# B&R Automation Studio project TD52 (part 130)

#### op_stateCyclic.st - OpState task
```iecst
(*******************************************************************************
AGGR: selection of the operating state (cyclic)

This code is confidential AND proprietary to the INNIO Company.
It may not be used in any form, or reproduced in any manner, without the express
written permission of the INNIO Company.
Copyright, INNIO Company, 2023

Customized modifications: -
------------------------
- Calculation of actual power in kW and permill
- Filtering of actual power
- Selection of the operating state of the engine in dependence of
  speed (n_ist) generator switch (gen_sch) and mains switch (net_sch)
- Creating of operating message for the alarmmanagement

History:
-------
V0.1	13-06-2001	Fahringer, generated from betr_zus V0.2
		20-07-2001	Fahringer, last modification
V0.2	03-09-2002	Fahringer, clculation of n_ist, p_ist, P_IST_OF,
							   ssPowerEx, P_IST_PROM add
V0.3	26-10-2002	Fahringer, engine speed meassured via ignition system
V0.31	21-11-2003	Fahringer, 100 rpm hystersis between StartM and LeerlM
V0.4	18-04-2004	Fahringer, calculation of speed is done in eng_ctr
V0.5	12-02-2007	Weitzer,   copy DIs for GCB and MCB to existiong PVs
							   replace mA power input by ssPAct from MMUSynch
V0.51	18.01.2008	Lechner,   adapted net_sch for test-bench run
V0.52	30.09.2010	Maier (BuR),	allocation DI_GCB_ON_TC1 to gen_sch deleted
		30.09.2010	Maier (BuR),	gen_sch replaced with GCB_ON_TC1
		01.10.2010	Maier (BuR), 	net_sch replaced with bPowerMode
		01.10.2010	Maier (BuR),	DI_MCB_ON_TC1 replaced with MCB_ON_TC1

--------------------
V3.99.0	19.10.2011	Graus,		implementation of the module for modular software
V3.99.1	24.10.2012	Graus,		extension of early opening of gas valves
V3.99.2	07.11.2012	Graus,		upgrade opstate machine function
								start state only is activated in transition from stop state
V3.99.3	12.11.2012	Graus,		change PT of xTOF_OpHour to T#10s
					Ze			AND NOT M_ABLOCK; 	 *changed, 4.6.13*
		18.11.2013	Graus,		bugfix FOR possible division BY 0
		17.12.2013	Graus,		bugfix - use case for OMSS and RSS state instead of direct comparisons in logic terms
V3.99.4 29.01.2014 	zengerer	bGV_Start_ScaveBlock Interface
V4.00.0 11.02.2014 	Graus,		change Version TO 4.0
V4.00.1 06.03.2014 	Graus,		change name of bGlowIgnPrevent to bGlowIgnPrevActive
V4.00.2 30.04.2014	Graus, Ze	M_ABLOCK := NOT(
V4.01.0 19.05.2014  Denk		Bugfix. Abstellstörung 1023 wie bei XT4 Pilotanlage
								Blockierung mit N_OP.tDI_Dem_EU_Block.Di
V4.01.1 27.05.2014  Graus		Delay FOR OMSS states like in XT3 (T=1s)
								Bugfix FOR bEng_Bloc
V4.01.2 27.05.2014  Graus		add bLockAckStarter to blocking engine
V4.01.3 02.06.2014	Weitzer		logic of M_ABLOCK corrected
					Denk/Weitzer block engine by EVU corrected
V4.01.4 24.06.2014  Graus		add bEng_Bloc_SGM(M_GM_Ref) to opstate logic
V4.01.5	15.10.2014	Caks,		added glow ignition, blocks module after run
V4.01.6	27.11.2014	Graus,		add submode TO opstate status
V4.02.0	24.02.2015	Graus,		add changes for J920 blocking engine
V4.02.1 13.03.2015	Graus,		bugfix: invert usage of IN_OP.bEng_Bloc_EC for bEng_Bloc
		20.10.2015	Caks,		added counters for: demand, netp and island operation
V4.03BETA 15.12.	Zengerer	new State 32: waiing for next automatic start (for new BR4 start procedure)
V4.03	26.01.2016	Perktold	changed bEng_Block_EVU in case of manual mode
V4.04.00	11.10.2016	Gwiggner	change Version TO 4.04
			19.10.2016	Gomez Ortiz	Modification of the cooling run phase
			28.10.2016	Gomez Ortiz	Separation between engine operation hour counter and unit op. hour counter
			21.12.2016  Denk		Modification for WinMOD simulation

 			02.02.2016	Zengerer	Modification for state 32 waiting for next automatic start
 			02.02.2017	lettenb.	OUT_OP.bEng_Bloc: ...FC_Rdy included(sky)
V4.05.00	24.04.2017	Denk		SWAT 920 Rel.2, block engine after 5 times W2462
			10.05.2017	Gomez Ortiz	Changes for Spezifikation_Ölkreislauf_Schnellstart_BR9
			14.06.2017	lettenb.	ZM_M_REL: bRelEngStart_OilSkid added acc.spec.gen.oilskid, xGR_MAXR_OpenGV.Gw:= 80->60 for 920(fahringer)
			26.06.2017	lettenb.	tEng_Aux_Dem_CDR2/3 added for multiple use(grain)
			10.07.2017	Denk		SWAT 920 Rel.3, block engine after 5 times W2465
			31.07.2017  Denk		SWAT 920, changes after validation. Deflagration protection different function for type 6 and type 9
			07.11.2017  Perktold,	op_state Task changed for houseload requirement
			19.01.2018	Gomez Ortiz	Extension of the early open valve timing for type 9 engines
			09.02.2018	Perktold	920er FastStart change for OUT_OP.tEng_Aux_Dem_CDR.Do calculation - bFS_Act deleted
V4.05.02	05-04-2018	Perktold,	added IN_OP.bFS_Act for OilSkid Start Release Type 9
V4.05.03	05-09-2018	Gwiggner	BU 01: bugfix function block xTP_OpenGV
V4.06.00	12-06-2018	Perktold	changes for GEN2/FastStart
V4.06.01	18.09.2018	Zengerer	new engine blocking at W1995 Perm Error
			03-10-2018	Hohensinner	Bugfix: Engine ready remote only when synchronization selector switch in position automatic
V4.07.00	25.04.2018	lettenb.	1165,9214 start lockout added, SWAT920/5
			14.01.2019	Schmid		W9249 (deflagration detection) blocks engine restart
V4.07.01	30.01.2019	Hohensinner	Code clean up and Diagnose Interfaces
			03.02.2019	Perktold	tEng_Run.Do geändert (BugFix)
			25.02.2019	lettenb.	bERV_NotRdy added, engine room ventilation not ready - block engine start, PWR-FFI-2018-0637 gem. TA 1100-0110
			13.03.2019	Hohensinner	block engine at low EO/ECW temperatures for type9, block engine at grid code data structure failure
V4.07.04	10.04.2019	Hohensinner	removed UPS DI signals from engine blocked array & cleanup #07
V4.07.05	15.05.2019	Hohensinner	added EngBlock_PlantCtr DI --> Blocks module smooth
			20.05.2019	Hohensinner	EngBlock_PlantCtr DI debugged for smooth shutdown in manual mode
			04.11.2019	Schmidt		BU 01: Type 6 cooldown run duration modified from 0s to 10s
V4.09.00	28.11.2019	lettenb.	bBloc_SY_ProtTest added, protection test(ThJ)
			13.01.2020	Arnold,		time delay for early GV opening changed to 9.8s
			12.02.2020	Zuschnig, 	included B2972 and B2973 - Power Mode on/off
V4.10.00	22.05.2020	lettenb.	bEng_Bloc[29-33] added
			20.10.2020	Zuschnig,	removed activation of module blocked by oil skid only if fast start is active -> always active
			16.10.2020	Weitzer,	release power mode by customer bit bReq_PowMod_Ext
			07.10.2020	Perktold	added fast start counter
			18.01.2021	Perktold	unbundling emergency stop and fire alarm
			18.01.2021	Weitzer		IN_OP.bBloc_SY_Rel_Cust to SY release array added
			27.01.2021  Zuschnig	Ensure TON,TOF,TP are always executed
V4.11.00	22.11.2021	Perktold,	added myPlant remote request/P-setpoint
			14.10.2021	Andre,		added SAFI in operation mode to start up release
			02.02.2022	Schmid,		no start blockade by ECWP_FC_Rdy in case of black start
V4.12.00	08.09.2022	Andre,		added SEMIC in operation mode to start up release
			20.09.2022	Perktold,	Additional delay for ignition deactivation for non-successful starts
			26.09.2022	Perktold,	Added IN signal to xTOFIgn_Dem in case of a prio 1 trip
			10.01.2023	lettenb.	bReq_Bloc[4]: bOMSS_MAN->(OUT_OP.iIdx_OMSS = 1), bOMSS_MAN is too slow for bumpless switchover MAN -> AUT, #966
			25.01.2023	Tinello		Added engine blocked by charge temperature after TC
V4.13.00	26.09.2023	Farre,		Addition engine blocked by LCB opened (info #37)
			24.08.2023	Zengerer	Add counter correction IN_OP.iCnt_OpHours_Set, iCnt_UnitOpHours_Set, iCnt_FastStarts_Set, iCnt_FastStarts_Set
			03.11.2023	Zuschnig	Add operating counter low load
			20.11.2023	Farre,		added "request power mode" interface from CU needed for Microgrid (2023-168)
			04.12.2023	Goenczi		Added Emergency request via Bus coupling - bEng_Dem_EPS_Bus
			04.12.2023	Goenczi		Hand over iIdx_Eng_State to OUT_OP
			17.01.2024	Schmidt		Bugfix deflagration protection: added IN_OP.bIgnDeflPrct_Off to ignition demand logic (issue 1406)
V4.14.00	28.03.2024	Soto/Farre,	Added CAN WG configuration for start up release (2023-174)
			25.10.2024	Farre		include in bEng_Bloc[1] - rel. sync- when GCB position signal failure and enigne stopped (2024-241)
			25.11.2024	Bacci		T6 Start procedure with purge start (2024-219): added waiting time for starter release in state 32 and 7

Instructions for use:
--------------------

Outstandings:
------------

*******************************************************************************)

FUNCTION AND_Array
	memcpy(ADR(Arrayx),Adress,MIN(40,Size) + 1);
	AND_Array	:=	 TRUE;
	FOR i:= 0 TO MIN(40,Size) DO
		AND_Array	:=	AND_Array AND Arrayx[i];
	END_FOR
END_FUNCTION

FUNCTION OR_Array
	memcpy(ADR(Arrayx),Adress,MIN(40,Size) + 1);
	OR_Array	:=	 FALSE;
	FOR i:= 0 TO MIN(40,Size) DO
		OR_Array	:=	OR_Array OR Arrayx[i];
	END_FOR
END_FUNCTION

FUNCTION DINT_INC_CNT
	DINT_INC_CNT	:=	Input + 1;
	IF DINT_INC_CNT >= 1000000000 THEN
		DINT_INC_CNT := DINT_INC_CNT - 1000000000;		(* check upper limit *)
	ELSIF DINT_INC_CNT <= -1000000000 THEN
		DINT_INC_CNT := DINT_INC_CNT + 1000000000;		(* check lower limit *)
	END_IF;
END_FUNCTION

PROGRAM _CYCLIC

(** 1: Execute EngType for Module *)
	xEngType.Motortype := INT_TO_UINT(Para.iEng_Motortype);
	xEngType();

(** 2: Build OMSS and RSS bits for states *)
	xTOF_OFF(IN := OUT_OP.iIdx_OMSS = 0, PT := T#1s);
	xTOF_MAN(IN := OUT_OP.iIdx_OMSS = 1, PT := T#1s);
	xTOF_AUTO(IN := OUT_OP.iIdx_OMSS = 2, PT := T#1s);
	xTOF_TEST(IN := OUT_OP.iIdx_OMSS = 3, PT := T#1s);
	xTOF_SCAV(IN := OUT_OP.iIdx_OMSS = 4, PT := T#1s);
	xTON_Eng_SU_Aut(IN := OUT_OP.bEng_SU_Aut, PT := T#6s);  (*V4.04 -> State 32*)

	bOMSS_OFF := xTOF_OFF.Q;
	bOMSS_MAN := xTOF_MAN.Q;
	bOMSS_AUTO := xTOF_AUTO.Q;
	bOMSS_TEST := xTOF_TEST.Q;
	bOMSS_SCAV := xTOF_SCAV.Q;

	bRSS_OFF := OUT_OP.iIdx_RSS = 0;
	bRSS_ON  := OUT_OP.iIdx_RSS = 1;
	bRSS_REM := OUT_OP.iIdx_RSS = 2;

	OUT_OP.tOMSS_MAT.Do := bOMSS_MAN OR bOMSS_AUTO OR bOMSS_TEST;

(** 3: Reject to house load type 6 / Fangen im Eigenbedarf Baureihe 6*)
	bTrigger_Island	:= xEngType.Type6 AND Para.bRej2houseload AND xOpMode.NetP AND (IN_OP.rN_EngAct >= rN_Eng_Limit);
	TOF_bTrigger_Island(IN := bTrigger_Island, PT := tOff_Trigger);

(** 4: Powermode *)
	bPowerMode := ((IN_OP.tMCB_On.Di AND NOT TOF_bTrigger_Island.Q) AND (IN_OP.tMnsOk.Di OR NOT IN_OP.bTestBenchModeIsland)) OR IN_OP.bReq_PowMod OR IN_OP.bReq_PowMod_Ext;

	IF IN_OP.tGCB_On.Di AND OUT_OP.tEng_Run.Do AND NOT IN_OP.tMCB_On.Di AND NOT IN_OP.bMCB_DemSy AND (IN_OP.bReq_PowMod OR IN_OP.bReq_PowMod_Ext) AND NOT bMsg2973 THEN
		bMsg2972 := TRUE;
	ELSE
		bMsg2972 := FALSE;
	END_IF;

	TOF_b2973(IN := EDGENEG (bMsg2972), PT := T#5s);
	bMsg2973 := TOF_b2973.Q;

(** 5: OpMode State machine: condition of engine state in dependence of actual speed, generator switch and mains switch*)
	IF IN_OP.rN_EngAct < 50 THEN							(* condition for engine operating state STOP	*)
		OUT_OP.iSt_OpMode := 16#00010000 * 10;	(* StopM -> 10 *)
	ELSE
		IF xOpMode.Stop THEN (* transition from stop mode *)
			bStop2Start := TRUE;
		END_IF;
		IF (IN_OP.rN_EngAct < Para.rN_Start_Trig) AND bStop2Start THEN			(* condition for engine operating state START	*)
			OUT_OP.iSt_OpMode := 16#00010000 * 30;	(* StartM -> 30 *)
		ELSE
			bStop2Start := FALSE;
			IF IN_OP.tGCB_On.Di AND bPowerMode THEN		(* condition for engine operating in parallel with system	*)
				OUT_OP.iSt_OpMode := 16#00010000 * 50;	(* NetpM -> 50 *)
			ELSE
				IF IN_OP.tGCB_On.Di AND NOT bPowerMode THEN	(* condition for engine operating in isolated mode	*)
					OUT_OP.iSt_OpMode := 16#00010000 * 60;	(* InselM -> 60 *)
				ELSIF IN_OP.rN_EngAct >= Para.rN_Start_Trig THEN
					OUT_OP.iSt_OpMode := 16#00010000 * 40;	(* LeerlM -> 40 *)
				END_IF;
			END_IF;
		END_IF;
	END_IF;

	xOpMode(in := OUT_OP.iSt_OpMode);

(** 6: Emergency Request *)
	OUT_OP.bEng_Dem_EPS	:=
							((IN_OP.tEng_Dem_EPS_Ext.Di OR IN_OP.bEng_Dem_EPS_Bus OR IN_OP.bEng_Dem_EPS_Sy) AND NOT IN_OP.bOnly_Island)
						OR 	(IN_OP.bOnly_Island AND NOT IN_OP.bOtherGenParallel);

	xTOF_EngDemEPS(IN:= OUT_OP.bEng_Dem_EPS AND NOT IN_OP.tGCB_On.Di, PT:= T#60s);
	bNoMon4BlackStart := xTOF_EngDemEPS.Q AND OUT_OP.bEng_Dem_EPS; //T14

(** 7: Excitation bit *)
	OUT_OP.bEng_SUpE := IN_OP.tEng_SUExc_Rel.Di;

(** 8: Plant control *)
	(** 8.1: W1188 release by station missing *)
	xTP_AT27(IN := NOT IN_OP.tRel_MasCtr.Di, PT := T#300s);
	AT27	:=	NOT xTP_AT27.Q AND IN_OP.tRel_MasCtr.Di;

	(** 8.2: Wxxxx block by plant control - smooth *)
	xTON_Block_PlantCtr(IN:= IN_OP.tEngBlock_PlantCtr.Di AND IN_OP.tEngBlock_PlantCtr.GoodQual, PT:=T#100ms);
	bEng_Block_PlantCtr	:=	xTON_Block_PlantCtr.Q;

	IF bEng_Block_PlantCtr AND bOMSS_MAN THEN																	(* set load to zero in manual mode *)
		VIS2MM.rP_set_vis		:=	0;
	END_IF
	IF EDGEPOS(bEng_Block_PlantCtr AND bOMSS_MAN AND (OUT_OP.rP_Act_Norm_Filt < 0.1 OR xOpMode.Island)) THEN	(* stop engine if under 10% load or island mode *)
		OUT_OP.bEng_Stop_Man	:=	TRUE;
	END_IF

(** 9: Engine Blocked Array  *)
	(* Info compared to old SW: 0-7 represents old variable "NOT ZM_M_REL" *)
	bEng_Bloc[0]	:=	NOT ((IN_OP.bMainsReturn AND (IN_OP.bRelMainsConnect OR xOpMode.NetP)) OR IN_OP.bRel_Island OR IN_OP.bRel_IslandAfMITime OR NOT Para.bSyActive);	(* Mains failure *)
	bEng_Bloc[1]	:=	(NOT IN_OP.bRelEngOpFromSy) OR IN_OP.bGCB_psf_EngStop;																								(* Release from Sync missing or gcb position failure when engine stopped *)
	bEng_Bloc[2]	:=	NOT AT27 OR (bEng_Block_PlantCtr AND NOT bEng_StaSpdExc);																							(* W1188 release by station missing *)
	bEng_Bloc[3]	:=	NOT IN_OP.bGasSupplyOk;																																(* Gas supply missing *)
	bEng_Bloc[4]	:=	NOT (	(NOT xEngType.Type9 AND NOT IN_OP.bDeflagrationPrct)																						(* Deflagration protection not Type 9 *)
							OR	(xEngType.Type9 AND ((NOT IN_OP.bDeflagrationPrct AND NOT IN_OP.bPBC_Active) OR IN_OP.bPBC_Active)));										(* Deflagration protection Type 9 *)
	bEng_Bloc[5]	:=	NOT IN_OP.tGV_Rel.Do;																																(* Gas valve release missing *)
	bEng_Bloc[6]	:=	IN_OP.bLockAckStarter;																																(* Starter temperature *)
	bEng_Bloc[7]	:=	xEngType.Type9 AND NOT bEng_StaSpdExc AND NOT IN_OP.bRelEngStart_OilSkid;																			(* Oil skid Type 9 *)
	bEng_Bloc[8]	:=	IN_OP.bEng_Block_Customized;																														(* Customer specific *)
	bEng_Bloc[9]	:=	IN_OP.tMCB_On.Di AND NOT OUT_OP.tEng_Run.Do AND IN_OP.tP_GenC_Bloc.Do;																				(* EU - Power reduction over limit *)
	bEng_Bloc[10]	:=	(IN_OP.bMsg3583 OR 	IN_OP.bMsg3584) AND Para.bGlowIgnPrevActive;																					(* Special gas: Exhaust gas temperatures *)
	bEng_Bloc[11]	:=	IN_OP.bSG_Eng_Block_EGT; 																															(* Special gas: blocked after 30min operation *)
	bEng_Bloc[12]	:=	IN_OP.bEng_Bloc_EC;(* AND Para.bSA_PI_Active;*)																										(* Blocked by Engine Controller*)
	bEng_Bloc[13]	:=	IN_OP.bSAFIPBCConfNotOK AND Para.bSA_PBC_Active;																									(* Blocked by SAFI PBC configuration *)
	bEng_Bloc[14]	:=	(bOMSS_AUTO AND NOT bEng_StaSpdExc AND NOT IN_OP.tScavFanFC_Rdy.Di);																				(* Blocked by FC scavanging fan *)
	bEng_Bloc[15]	:=	(bOMSS_AUTO AND NOT bEng_StaSpdExc AND NOT IN_OP.tECWP_FC_Rdy.Di AND NOT bNoMon4BlackStart);														(* Blocked by FC ECWP *)
	bEng_Bloc[16]	:=	(bOMSS_AUTO AND NOT bEng_StaSpdExc AND NOT IN_OP.tEOP_FC_Rdy.Di);																					(* Blocked by FC EOP *)
	bEng_Bloc[17]	:=	(bOMSS_AUTO AND NOT bEng_StaSpdExc AND NOT IN_OP.tBbBlower_FC_Rdy.Di);																				(* Blocked by FC Byblower *)
	bEng_Bloc[18]	:=	((IN_OP.bAMM_Pr_MGT_a_Filt_BlockStart OR IN_OP.bAMM_Pr_PCGT_a_Filt_BlockStart) AND xEngType.Type9); 												(* 5times MSF in gastrain *)
	bEng_Bloc[19]	:=	(IN_OP.bMsg9214 AND NOT bEng_StaSpdExc AND xEngType.Type9); //SWAT920/5																				(* Engine turn equipment active *)
	bEng_Bloc[20]	:=	(IN_OP.bMsg1165 AND NOT bEng_StaSpdExc AND xEngType.Type9); //SWAT920/5																				(* Exhaust gas scavanging failure *)
	bEng_Bloc[21]	:=	(IN_OP.bMsg1995 AND NOT bEng_StaSpdExc );																											(* Perm failure in stop mode *)
	bEng_Bloc[22]	:=	IN_OP.tMCB_On.Di AND NOT OUT_OP.tEng_Run.Do AND IN_OP.tDI_Dem_EU_Block.Di;																			(* EU - Blocked by DI *)
	bEng_Bloc[23]	:=	IN_OP.tMCB_On.Di AND NOT OUT_OP.tEng_Run.Do AND IN_OP.bEng_Block_EVU;																				(* EU - Blocked by Bus *)
	bEng_Bloc[24]	:=	IN_OP.bMsg9249 AND NOT bEng_StaSpdExc;																												(* Deflagration detection *)
	bEng_Bloc[25]	:=	IN_OP.bERV_NotRdy AND NOT bEng_StaSpdExc;																											(* engine room ventilation not ready *)
	bEng_Bloc[26]	:=	xEngType.Type9 AND bOMSS_MAN AND NOT bEng_StaSpdExc AND IN_OP.bMsg2524;																				(* Type9: EO Temp low *)
	bEng_Bloc[27]	:=	xEngType.Type9 AND bOMSS_MAN AND NOT bEng_StaSpdExc AND bT_ECW_Lo;																					(* Type9: ECW Temp low *)
	bEng_Bloc[28]	:=	IN_OP.bEng_Bloc_GR AND NOT bEng_StaSpdExc;																											(* GR - data structure failure *)
	bEng_Bloc[29]	:=	NOT IN_OP.tScavFanCB_trip.Di AND NOT bEng_StaSpdExc;																								(* Blocked by CB scavenging fan tripped *)
	bEng_Bloc[30]	:=	NOT IN_OP.tGenIF_CB_On.Di AND NOT bEng_StaSpdExc;																									(* Blocked by CB generator interface panel tripped *)
	bEng_Bloc[31]	:=	IN_OP.bAMM_OilSkid_PumpLP_CB AND NOT bEng_StaSpdExc AND xEngType.Type9;																				(* Type9: Blocked by CB oil skid LP oil pump tripped *)
	bEng_Bloc[32]	:=	IN_OP.bAMM_OilSkid_PumpHP_CB AND NOT bEng_StaSpdExc AND xEngType.Type9;																				(* Type9: Blocked by CB oil skid HP oil pump tripped *)
	bEng_Bloc[33]	:=	IN_OP.bAMM_OilSkid_MCB AND NOT bEng_StaSpdExc AND xEngType.Type9;																					(* Type9: Blocked by oil skid main switch auxiliaries opened *)
	bEng_Bloc[34]	:=	NOT IN_OP.tECWP_CB_On.Di AND NOT bEng_StaSpdExc;																									(* Blocked by CB ECWP tripped *)
	bEng_Bloc[35]	:=	IN_OP.bEngBloc_EX AND NOT bEng_StaSpdExc;
	bEng_Bloc[36]	:=	NOT IN_OP.bRelEngStart_Ch_T2 AND NOT bEng_StaSpdExc;																								(* Blocked by charge temperature after TC *)
	bEng_Bloc[37]	:=	NOT IN_OP.tLineCB_On.Di AND IN_OP.tLineCB_On.GoodQual;																								(* Blocked by line circuit breaker open *)
	bEng_Bloc[38]	:=	IN_OP.bBlock_WG_CAN_Conf;																															(* Blocked by wastegate configuration in progress *)

	OUT_OP.bEng_Bloc		:=	OR_Array(ADR(bEng_Bloc),50);	(* 1 = engine is blocked *)
	MM2VIS.bEng_Bloc		:=	bEng_Bloc;						(* Array to VIS *)
	MM2VIS.bEng_Bloc_Show	:=	(iIdx_Eng_State = 19);			(* Show Array only on HMI if engine is blocked *)

(** 10: Demand Auxiliaries  *)
	OUT_OP.bEng_Aux_Dem :=	(OUT_OP.bEng_Dem AND (IN_OP.bPurgeER_Rdy OR NOT Para.bPurgecycle_Active) AND (IN_OP.bEGScav_Rdy OR OUT_OP.bEng_Dem_EPS)) OR IN_OP.bGV_On;

(** 11: Release Engine *)
	OUT_OP.bEng_Rel :=	OUT_OP.tOMSS_MAT.Do
						AND ((NOT (bGnlTrip1 OR bGnlTrip2 OR bGnlTrip3)) OR bDryTestBench)
						AND IN_OP.tPB2MM.bParaSetupOk;

(** 12: Start Up Release - Array for Manual and Automatic Mode *)
	bEng_SU[0]	:=	OUT_OP.bEng_Rel;																		(* Engine released *)
	bEng_SU[1]	:=	NOT bEng_StaSpdExc;																		(* Start speed not exceeded *)
	bEng_SU[2]	:=	IN_OP.bRelEngOp_Aux;																	(* Release from Auxiliaries *)
	bEng_SU[3]	:=	IN_OP.bScavFinished;																	(* Scavanging finished *)
	bEng_SU[4]	:=	(IN_OP.bPurgeER_Rdy AND IN_OP.tRel_ER_PurgeCycle.Di) OR NOT Para.bPurgecycle_Active;	(* Purge finished *)
	bEng_SU[5]	:=	NOT IN_OP.bEng_Bloc_SGM;																(* Special gas mixer calibration routine not active *)
	bEng_SU[6]	:=	IN_OP.bIC_OperationState AND IN_OP.bSA_CfgDone;											(* SEMIC used and in operation state *)

	MM2VIS.bEng_SU			:=	bEng_SU;																	(* Array to VIS *)
	MM2VIS.bEng_SU_Show		:=	(iIdx_Eng_State = 32) OR (iIdx_Eng_State = 9) OR (iIdx_Eng_State = 8) OR (iIdx_Eng_State = 6);	(* Show Array only on HMI if in this states *)

(** 13: Engine Ready Manual Mode *)
	OUT_OP.bEng_Rdy_Man :=	OUT_OP.bEng_Rel AND bOMSS_MAN AND NOT bEng_StaSpdExc AND NOT OUT_OP.bEng_Bloc;

(** 14: Start Impulse 10s long *)
	xTP_Imp_Start(IN := IN_OP.bEng_Start, PT := T#10s);
	OUT_OP.bImp_Start := xTP_Imp_Start.Q;

(** 15: Delay next manual start for 5s *)
	xTOF_BlocDelay_ManStart(IN := OUT_OP.bImp_Start OR IN_OP.bEng_Start , PT := T#5s);
	OUT_OP.bBlocDelay_ManStart := xTOF_BlocDelay_ManStart.Q;

(** 16: Blocking demand for 30s after a Start *)
	xTOF_ANFBLO(IN := bEng_StaSpdExc, PT := T#30s);
	OUT_OP.bEng_Dem_Bloc := xTOF_ANFBLO.Q;

(** 17: Start Up Failure - Manual Mode *)
	OUT_OP.bEng_Dem_Man_SUpF :=
							(bStart OR ZM_H_ANF OR OUT_OP.bEng_Dem_Aut OR (bOMSS_AUTO AND OUT_OP.bEng_CDR))
						AND OUT_OP.bEng_Rel
						AND bOMSS_MAN
						AND NOT OUT_OP.bEng_Stop_Man
						AND NOT OUT_OP.bEng_Bloc;

	ZM_H_ANF :=				OUT_OP.bEng_Dem_Man_SUpF
						AND (NOT OUT_OP.bEng_Dem_Bloc OR IN_OP.bGV_On OR IN_OP.bEng_Start);

(** 18: Engine Demand - Manual Mode *)
	OUT_OP.bEng_Dem_Man :=
						(NOT bStart OR OUT_OP.bEng_Dem_Man)
						AND ZM_H_ANF;

(** 19: Start Up Release - Manual Mode *)
	OUT_OP.bEng_SU_Man	:=	AND_Array(ADR(bEng_SU),6) AND OUT_OP.bEng_Dem_Man;			(* 1 = start up *)

(** 19: Engine Start up - Manual Mode *)
	OUT_OP.bEng_Rel_SU	:=	OUT_OP.bEng_SU_Man AND (NOT OUT_OP.bBlocDelay_ManStart OR IN_OP.bEng_Start);

(** 20: Notstrom Anforderung ohne reine Inselanlagen *)
	bRequest_EPS	:=	OUT_OP.bEng_Dem_EPS AND NOT IN_OP.bOnly_Island;				(* EPS *)

(** 21: Engine automatic request *)
	(** 21.1: Engine in Automatic demanded *)
	bReq_Dem[0]		:=	bRSS_ON;																	(* ON *)
	bReq_Dem[1]		:=	bRSS_REM AND VIS2MM.bRemoteReq AND Para.bRemoteReqActive;					(* HMI Button *)
	bReq_Dem[2]		:=	bRSS_REM AND IN_OP.tReq_PeakLoad.Di;										(* DI - Peakload *)
	bReq_Dem[3]		:=	bRSS_REM AND IN_OP.bBus_Dem;												(* BUS *)
	bReq_Dem[4]		:=	bRSS_REM AND IN_OP.bEngDSS_Mains;											(* Mains control *)
	bReq_Dem[5]		:=	bRSS_REM AND IN_OP.bCust_Dem;												(* Demand from Custom Module *)
	bReq_Dem[6]		:=	bRSS_REM AND IN_OP.tDemEngOpExt.Di;											(* DI - ExtDem *)
	bReq_Dem[7]		:=	bRSS_REM AND VIS2MM.bRemoteReq_myPlant AND Para.bRemoteReqMyPlantActive;	(* myPlant *)

	bReq_Remote		:= bReq_Dem[1] OR bReq_Dem[7];													(* Engine Demand via remote (HMI or myPlant) *)

	bRequest_Dem	:=	OR_Array(ADR(bReq_Dem),7);
	MM2VIS.bReq_Dem		:=	bReq_Dem;
	MM2VIS.bReq_Dem_Show:=	TRUE;		(* not used at moment *)

	(** 21.2: Block Automatic Engine demand *)
	bReq_Bloc[0]	:=	IN_OP.bGT_DemRelGasTypSwh; 									(* Gas type switching *)
	bReq_Bloc[1]	:=	IN_OP.tP_GenC_Bloc.Do;										(* EU load reduction > limit *)		//EVU_BLOCK_INT	Mathias 2.6.2014
	bReq_Bloc[2]	:=	IN_OP.tDI_Dem_EU_Block.Di;									(* EU - DI *)						//DI_EVU_BLOCK  Mathias 2.6.2014
	bReq_Bloc[3]	:=	IN_OP.bEng_Block_EVU;										(* EU - Bus *)
	bReq_Bloc[4]	:=	bRequest_EPS AND (OUT_OP.iIdx_OMSS = 1);					(* EPS & OMSS Man *)
	bReq_Bloc[5]	:=	bRequest_EPS AND IN_OP.bSmoothDischarge;					(* EPS & smooth discharge *)
	bReq_Bloc[6]	:=	bEng_Block_PlantCtr;										(* PlantCtr *)

	bRequest_Bloc	:=	OR_Array(ADR(bReq_Bloc),6);
	MM2VIS.bReq_Bloc:=	bReq_Bloc;
	MM2VIS.bReq_Bloc_Show	:=	TRUE;	(* not used at moment *)

	(** 21.3: Request Engine - M_ANF *)
	xTON_T105(IN := bOMSS_TEST AND (xTON_T105.Q OR OUT_OP.tEng_Run.Do), PT := T#300s);	(* Test delay *)

	bReq_A[0] 		:=	bRequest_Dem AND NOT bRequest_Bloc;								(* Requested and not blocked *)
	bReq_A[1] 		:=	bRequest_EPS AND NOT IN_OP.bSmoothDischarge AND NOT bOMSS_MAN AND NOT bEng_Block_PlantCtr;	(* EPS request *)
	bReq_A[2] 		:=	bOMSS_MAN AND IN_OP.tGCB_On.Di;									(* OMSS Man and GCB closed *)
	bReq_A[3] 		:=	bOMSS_TEST AND (NOT xTON_T105.Q OR IN_OP.tReq_Test.Di); 		(* OMSS Test and Test Delay / DI *)

	bRequest_A 		:=	OR_Array(ADR(bReq_A),3);
	MM2VIS.bReq_A	:=	bReq_A;
	MM2VIS.bReq_A_Show	:=	bOMSS_AUTO;

	M_ANF	:= 	bRequest_A; 	(* rückwärtskompatiblität *)

(** 22: Engine demand start up failure & Engine demand in automatic mode *)
	xGRMinR_KWT(Gw := Para.rT_ECW_LimLo, Hy := Para.rT_ECW_HyLo, In := IN_OP.tT_ECW.Ai);
	xTON_kwtp(IN := xGRMinR_KWT.Q AND IN_OP.tPB2MM.bParaSetupOk, PT := T#2s);
	bT_ECW_Lo := xTON_kwtp.Q;	(* entspricht AN_KTMI - Kühlwassertemperatur minimum *)									//Überprüfen ob in powersel unten benötigt, vllt besser: von HC hermappen

	(* Release automatic start - M_ABLOCK *)
	bEng_Dem_A[0]	:=	NOT bT_ECW_Lo OR OUT_OP.bEng_Dem_EPS; 														(* Engine cooling water temperature not low *)
	bEng_Dem_A[1]	:=	NOT IN_OP.bPr_N2_LoTon OR OUT_OP.tEng_Run.Do OR IN_OP.bGT2_Select OR NOT IN_OP.bRel_ScavN2;	(* N2 scavanging done *)
	bEng_Dem_A[2]	:=	NOT OUT_OP.bEng_Bloc;																		(* Engine not blocked *)

	(* Release automatic start - OUT_OP.bEng_Dem_Aut_SUpF *)
	bEng_Dem_A[3]	:=	OUT_OP.bEng_Rel;																			(* Engine released *)
	bEng_Dem_A[4]	:=	bOMSS_AUTO OR bOMSS_TEST;																	(* OMSS Auto or Test *)
	bEng_Dem_A[5]	:=	bRequest_A;																					(* Engine automatic start requested *)

	(* Release automatic start - OUT_OP.bEng_Dem_Aut*)
	bEng_Dem_A[6]	:=	NOT bEng_StaSpdExc OR IN_OP.bGV_On OR IN_OP.bEng_Start;										(* Engine starts / runs *)
	bEng_Dem_A[7]	:=	NOT OUT_OP.bEng_Dem_Bloc OR	OUT_OP.tEng_Run.Do OR OUT_OP.bEng_Dem_Aut;						(* Engine request blocked, before: M_ANFBLO *)
	bEng_Dem_A[8]	:=	NOT IN_OP.tERDF_BLOCK.Do;																	(* ERDF *)
	bEng_Dem_A[9]	:=	NOT IN_OP.bOpMsg_Plim_ERDF_ABF_SOnOf;														(* Load reduction over limit *)

	M_ABLOCK					:=	AND_Array(ADR(bEng_Dem_A),2); 	//M_ABLOCK wird nun im array gebildet, bildet sich nur aus 0 bis 2
	OUT_OP.bEng_Dem_Aut_SUpF	:=	AND_Array(ADR(bEng_Dem_A),5);	//OUT_OP.bEng_Dem_Aut_SUpF bildet sich nur aus 0 bis 5
	OUT_OP.bEng_Dem_Aut			:=	AND_Array(ADR(bEng_Dem_A),9);
	MM2VIS.bEng_Dem_A			:=	bEng_Dem_A;
	MM2VIS.bEng_Dem_A_Show		:=	bOMSS_AUTO;

	ZM_M_BERAUT :=			OUT_OP.bEng_Rel
						AND (bOMSS_AUTO OR (bOMSS_TEST AND OUT_OP.bEng_Dem_EPS));

(** 23: Engine ready for automatic mode *)
	OUT_OP.bEng_Rdy_Aut		:=	ZM_M_BERAUT AND M_ABLOCK; 	(*changed, 4.6.13*)

(** 24: Engine ready for automatic mode - info for exitation system *)
	OUT_OP.bEng_Rdy_Aut_Exc	:=	ZM_M_BERAUT	AND (bRequest_A OR NOT IN_OP.bOnly_Island);

(** 25: Engine ready for remote operation *)
	OUT_OP.tEng_Rdy_Rem.Do	:=	OUT_OP.bEng_Rdy_Aut AND bRSS_REM AND IN_OP.iIdx_SyOMSS = 2;

(** 26: Engine automatic startup *)
	OUT_OP.bEng_SU_Aut		:=	AND_Array(ADR(bEng_SU),6) AND OUT_OP.bEng_Dem_Aut;		(* 1 = start up *)

(** 27: Engine monitoring of after start for 10s *)
	xTOF_T9(IN := IN_OP.bEng_Start, PT := T#10s);
	OUT_OP.bEng_MonOff := xTOF_T9.Q;

(** 27: Engine stop in manuel mode *)
	OUT_OP.bEng_Stop_Man	:=	(OUT_OP.bEng_Rel AND bOMSS_MAN  AND bStop)
							OR	(OUT_OP.bEng_Rel AND bOMSS_MAN  AND OUT_OP.bEng_Bloc)
							OR	(OUT_OP.bEng_Rel AND bOMSS_MAN  AND NOT bEng_StaSpdExc AND IN_OP.bMaxPreLubeTime)
							OR	(OUT_OP.bEng_Rel AND bOMSS_AUTO AND IN_OP.bN_EngStartDrop)
							OR	(OUT_OP.bEng_Rel AND bIgn_DemTemp AND OUT_OP.bEng_Stop_Man);						//latch until ignition demand off

(** 28: Demand Ignition *)
	xTON_T_Z_AUS(IN := IN_OP.bMsg1026, PT := T#10s);

	bIgn_Dem[0]	:=	NOT IN_OP.bMsg1022 OR IN_OP.bIgn2_Sel;							(* A1022 - overspeed (relay)				*)
	bIgn_Dem[1]	:=	NOT bGnlTrip1 OR IN_OP.bIgn2_Sel;								(* Trip1									*)
	bIgn_Dem[2]	:=	NOT xTON_T_Z_AUS.Q;												(* A1026 - Shutdown failure, 10s delayed	*)
	bIgn_Dem[3]	:=	IN_OP.bRel_IgnOn OR bEng_StaSpdExc;								(* Release ignition from starter (AG)		*)
	bIgn_Dem[4]	:=	NOT IN_OP.bN2_ScavCoStarterOn OR NOT IN_OP.bRel_ScavN2;			(* N2 scavanging in progress				*)
	bIgn_Dem[5]	:=	NOT IN_OP.bIgnDeflPrct_Off;										(* Deflagration protection					*)

	bIgn_DemTemp	:=	AND_Array(ADR(bIgn_Dem),5) OR ((IN_OP.b_ST_DemIgn OR IN_OP.rN_EngAct <> 0) AND IN_OP.bSelfTestRunning);
	MM2VIS.bIgn_Dem	:=	bIgn_Dem;
	MM2VIS.bIgn_Dem_Show	:=	TRUE;

	(** 28.1: Demand Ignition off is delayed, only in case of priority 1 trip it is not delayed *)
	IF IN_OP.tAB2OP.bGnlTrip1 THEN
		OUT_OP.tIgn_Dem.Do := bIgn_DemTemp;
		xTOFIgn_Dem(IN:= bIgn_DemTemp);
	ELSIF NOT IN_OP.tAB2OP.bGnlTrip1 THEN
		IF bEng_StaSpdExc THEN
			xTOFIgn_Dem(IN:= bIgn_DemTemp, PT:= Ign_Dem_DelayTime);
		ELSE
			xTOFIgn_Dem(IN:= bIgn_DemTemp, PT:= Ign_Dem_DelayTime + Ign_Dem_DelayTime2);
		END_IF;
		OUT_OP.tIgn_Dem.Do := xTOFIgn_Dem.Q;
	END_IF;
	OUT_OP.bIgn_Dem	:=	OUT_OP.tIgn_Dem.Do;

(** 29: Demand gas valves *)
	(** 29.1: early opening of gas valves *)
	IF xEngType.Type9 THEN
		xGR_MAXR_OpenGV.Gw	:=	60;
		xTP_OpenGV.PT		:=	T#9s800ms;		(* Type 9 engine needs approx. 10 seconds for the ignition unit to be ready *)
	ELSE
		xGR_MAXR_OpenGV.Gw	:=	80;
		xTP_OpenGV.PT		:=	T#4s800ms;	(* Other engines need approx. 6 seconds for the ignition unit to be ready *)
    END_IF;
	xGR_MAXR_OpenGV(In := IN_OP.rN_EngAct, Hy := 10);
	xTP_OpenGV(IN:= xGR_MAXR_OpenGV.Q AND IN_OP.bEng_Start AND NOT Para.bGlowIgnPrevActive AND NOT Para.bDeAct_EarlyGV_opening AND (IN_OP.iStartCount = 1));

	(* 29.2: Release of gas valves *)
	OUT_OP.bGV_Rel :=		NOT IN_OP.bMsg1031
							AND NOT IN_OP.bMsg1054
							AND NOT IN_OP.bMsg1022
							AND NOT IN_OP.bMsg1026
							AND NOT bGnlTrip1;

	(* 29.3: Gas valves open *)
	bGV_Open[0] :=	OUT_OP.bEng_Rel OR (bGnlTrip3 AND (bOMSS_AUTO OR bOMSS_TEST));
	bGV_Open[1] :=	bIgn_DemTemp;
	bGV_Open[2] :=	IN_OP.bIgn_Run OR xTP_OpenGV.Q;
	bGV_Open[3] :=	NOT xOpMode.Stop;
	bGV_Open[4] :=	NOT OUT_OP.bEng_Stop_Man;
	bGV_Open[5] :=	OUT_OP.bGV_Rel;
	bGV_Open[6] :=	((	IN_OP.tN2_GV1_Closed.Di AND (IN_OP.tN2_GV2_Closed.Di OR NOT Para.bSel_TwoN2Valves) AND IN_OP.tScavVaClosed.Di) OR NOT IN_OP.bRel_ScavN2 OR IN_OP.bGV_On);
	bGV_Open[7] :=	NOT IN_OP.bGV_Start_ScaveBlock;	 (*new:	block gas valves from startup procedure	for scavening start *)

	OUT_OP.bGV_Open_Opstate	:=	AND_Array(ADR(bGV_Open),7);
	MM2VIS.bGV_Open			:=	bGV_Open;
	MM2VIS.bGV_Open_Show	:=	bIgn_DemTemp;

(** 30: Engine demand *)
	OUT_OP.bEng_Dem		:=	OUT_OP.bEng_Dem_Man
						OR	OUT_OP.bEng_Dem_Aut
						OR	OUT_OP.bEng_SUpE;

(** 31: RPS Demand *)
	OUT_OP.bEng_RPSDem	:=	OUT_OP.bEng_Dem
						AND NOT IN_OP.bGT_DemRelGasTypSwh
						AND (NOT bOMSS_TEST OR (bOMSS_TEST AND IN_OP.tReq_Test.Di) OR OUT_OP.bEng_Dem_EPS);

(** 32: Engine Cool down run *)
	ZM_IN_bEng_CDR	:=	OUT_OP.tEng_Run.Do
					AND ( 	((bOMSS_AUTO OR bOMSS_TEST) AND IN_OP.tGCB_On.Di)
						OR	OUT_OP.bEng_Dem_Aut
						);

	ZM_RS_bEng_CDR	:=	(NOT bOMSS_AUTO AND NOT bOMSS_TEST)
					OR	bGnlTrip1
					OR	bGnlTrip2
					OR 	OUT_OP.bEng_Bloc;

	IF xEngType.Type6 THEN
		xTOF_R_bEng_CDR(IN := ZM_IN_bEng_CDR, PT := 1000, RS := ZM_RS_bEng_CDR);  (* PT = 1000 -> Delaytime in 10ms steps -> 10s *)
	ELSIF xEngType.Type9 THEN
		xTOF_R_bEng_CDR(IN := ZM_IN_bEng_CDR, PT := 0, RS := ZM_RS_bEng_CDR);  (* PT = 0 -> Delaytime in 10ms steps -> 0s *)
	ELSE
		xTOF_R_bEng_CDR(IN := ZM_IN_bEng_CDR, PT := 6000, RS := ZM_RS_bEng_CDR);  (* PT = 6000 -> Delaytime in 10ms steps -> 6000s *)
	END_IF;

	OUT_OP.bEng_CDR := xTOF_R_bEng_CDR.Q;

(** 33: Engine run *)
	xGR_MAXR_bs_15s_rpm_hi(In := IN_OP.rN_EngAct, Gw := Para.rN_BS_Acc_LimHi, Hy := 10);
	bs_15s_rpm_hi :=
					xGR_MAXR_bs_15s_rpm_hi.Q
				AND IN_OP.tPB2MM.bParaSetupOk;
	bs_15s_rel_oper :=
					Para.bBS_Acc_Active
				AND OUT_OP.bEng_Dem_EPS
				AND OUT_OP.bEng_MonOff
				AND (bs_15s_rpm_hi OR bs_15s_rel_oper);

	IF (xOpMode.Idle OR xOpMode.Island OR xOpMode.NetP) AND NOT bN_Eng_Run THEN
		bN_Eng_Run	:= TRUE;
	ELSIF xOpMode.Stop AND bN_Eng_Run THEN
		bN_Eng_Run	:= FALSE;
	END_IF;

	OUT_OP.tEng_Run.Do :=
					OUT_OP.tOMSS_MAT.Do
				AND IN_OP.bGV_On
				AND ((bs_15s_rel_oper OR NOT OUT_OP.bEng_MonOff) OR bN_Eng_Run)	//Änderung >= rN_Start_Trig für Faststart schnellere SY
				AND (OUT_OP.bEng_CDR OR OUT_OP.bEng_Dem_Aut OR (bOMSS_MAN  AND OUT_OP.bEng_Dem_Man));

(** 34: Restart blocking *)
	xTON_RUN(IN := TRUE, PT := T#30s); (* instead RUN bit *)
	ZM_bEng_RSBoc	:=	(NOT OUT_OP.tEng_Run.Do AND xTON_RUN.Q)
					OR	EDGENEG(OUT_OP.tEng_Run.Do);

	xTP_bEng_RSBoc(IN := ZM_bEng_RSBoc, PT := T#2m);	// sinnvoller vieleicht nur auf EDGENEG gehen und das andere vergessen, dann wär es nur mehr bei echten abstellungen... nicht bei kaltstarts
	OUT_OP.bEng_RSBoc := xTP_bEng_RSBoc.Q;

(** 35: Gastypes *)
	OUT_OP.bGasTyp1_Act :=
						NOT IN_OP.bGT_Ipol12Active
					AND	(
							(IN_OP.bSelGasTyp1 AND (IN_OP.bLeanox_Man OR (NOT IN_OP.bGT_TypSwhActiveHalt AND NOT IN_OP.bGT_TypSwhActive AND NOT IN_OP.tSelGasTyp.Di)))
						OR	(
								((IN_OP.bGT_TypSwhActiveHalt AND NOT IN_OP.bGT2_Select) OR (IN_OP.bGT_TypSwhActive AND IN_OP.bGT_SelGas1) OR (IN_OP.tSelGasTyp.Di AND NOT IN_OP.tSelGasTyp2.Di AND NOT IN_OP.tSelGasTyp3.Di AND NOT IN_OP.tSelGasTyp4.Di))
							AND (NOT IN_OP.bLeanox_Man OR IN_OP.bSelGasTypAut)
							)
						);

	OUT_OP.bGasTyp2_Act :=
						(NOT IN_OP.bGT_Ipol12Active AND IN_OP.bSelGasTyp2 AND (IN_OP.bLeanox_Man OR (NOT IN_OP.bGT_TypSwhActiveHalt AND NOT IN_OP.bGT_TypSwhActive AND NOT IN_OP.tSelGasTyp.Di)))
					OR 	(
							((IN_OP.bGT_TypSwhActive AND IN_OP.bGT_SelGas2) OR (IN_OP.tSelGasTyp.Di AND IN_OP.tSelGasTyp2.Di AND NOT IN_OP.tSelGasTyp3.Di AND NOT IN_OP.tSelGasTyp4.Di))
						AND NOT IN_OP.bLeanox_Man
						);

	OUT_OP.bGasTyp3_Act :=
						(IN_OP.bSelGasTyp3 AND (IN_OP.bLeanox_Man OR (NOT IN_OP.bGT_TypSwhActiveHalt AND NOT IN_OP.bGT_TypSwhActive AND NOT IN_OP.tSelGasTyp.Di)))
					OR	(
							((IN_OP.bGT_TypSwhActiveHalt AND IN_OP.bGT2_Select) OR (IN_OP.bGT_TypSwhActive AND IN_OP.bGT_SelGas3) OR (IN_OP.tSelGasTyp.Di AND IN_OP.tSelGasTyp3.Di AND NOT IN_OP.tSelGasTyp4.Di))
						AND (NOT IN_OP.bLeanox_Man OR IN_OP.bSelGasTypAut)
						);

	OUT_OP.bGasTyp4_Act :=
						(IN_OP.bSelGasTyp4 AND (IN_OP.bLeanox_Man OR (NOT IN_OP.bGT_TypSwhActiveHalt AND NOT IN_OP.bGT_TypSwhActive AND NOT IN_OP.tSelGasTyp.Di)))
					OR	(
							((IN_OP.bGT_TypSwhActive AND IN_OP.bGT_SelGas4) OR (IN_OP.tSelGasTyp.Di AND IN_OP.tSelGasTyp4.Di))
						AND NOT IN_OP.bLeanox_Man
						);

	OUT_OP.bGasTypMix1_2_Act :=	IN_OP.bGT_Ipol12Active;

(** 36: start speed exceeded *)
	xGR_MAXR_Eng_StaSpdExc(In := IN_OP.rN_EngAct, Gw := Para.rN_EngStart_LimHi, Hy := Para.rN_EngStart_HyHi);
	xTOF_Eng_StaSpdExc(IN := xGR_MAXR_Eng_StaSpdExc.Q AND IN_OP.tPB2MM.bParaSetupOk, PT := T#10s);
	bEng_StaSpdExc := xTOF_Eng_StaSpdExc.Q;

(** 37: various demands of auxiliaries *)
	xTOF_Eng_Aux_Dem(IN := bEng_StaSpdExc OR OUT_OP.bEng_Aux_Dem, PT := T#300s);
	OUT_OP.bEng_Aux_Dem_TOF := xTOF_Eng_Aux_Dem.Q;
	OUT_OP.tEng_Aux_Dem_CDR.Do := OUT_OP.bEng_Aux_Dem_TOF AND (bEng_StaSpdExc OR (OUT_OP.tOMSS_MAT.Do AND NOT IN_OP.bMsg1031 AND NOT IN_OP.bMsg1054));
	OUT_OP.bEng_Aux_Dem_CDR	:= OUT_OP.tEng_Aux_Dem_CDR2.Do := OUT_OP.tEng_Aux_Dem_CDR3.Do := OUT_OP.tEng_Aux_Dem_CDR.Do;

(** 38: synchronization / load release *)
	xTOF_SoftShutdown(IN := IN_OP.bGV_On AND NOT bGnlTrip2, PT := T#1s);
	xGR_MINR_P_Lo(In:= OUT_OP.rP_Act_Norm, Gw:= Para.rP_LimLo, Hy:= Para.rP_HyLo);
	bP_Lo  := IN_OP.tPB2MM.bParaSetupOk AND xGR_MINR_P_Lo.Q;

	bSync_Rel[0]	:=	OUT_OP.tOMSS_MAT.Do;
	bSync_Rel[1]	:=	((IN_OP.bT_EOP_RelLoad OR NOT xEngType.Type9) AND IN_OP.bT_ECW_RelLoad AND NOT IN_OP.bT_ECW_Hi)
					OR	bOMSS_MAN
					OR	OUT_OP.bEng_Dem_EPS
					OR	IN_OP.tGCB_On.Di;
	bSync_Rel[2]	:=	OUT_OP.tEng_Run.Do
					OR 	(bGnlTrip2 AND xTOF_SoftShutdown.Q AND bOMSS_AUTO)
					OR 	(OUT_OP.bEng_SUpE  AND NOT bGnlTrip2 AND NOT bGnlTrip3);
	bSync_Rel[3]	:=	xTOF_SoftShutdown.Q OR	OUT_OP.bEng_SUpE;
	bSync_Rel[4]	:=	NOT bP_Lo OR NOT bGnlTrip2;
	bSync_Rel[5]	:=	NOT bGnlTrip1;
	bSync_Rel[6]	:=	NOT bOMSS_TEST
					OR 	(bOMSS_TEST AND IN_OP.tReq_Test.Di)
					OR 	OUT_OP.bEng_Dem_EPS
					OR 	IN_OP.tGCB_On.Di;
	bSync_Rel[7]	:=	NOT IN_OP.bMsg1218;
	bSync_Rel[8]	:=	IN_OP.tGV_Rel.Do;
	bSync_Rel[9]	:=	IN_OP.bsy_lfg_SG;
	bSync_Rel[10]	:=	NOT IN_OP.bBloc_SY_FS;
	bSync_Rel[11]	:=	NOT IN_OP.bBloc_SY_ProtTest;
	bSync_Rel[12]	:=	NOT IN_OP.bBloc_SY_Rel_Cust;
	bSync_Rel[13]	:=	TRUE;
	bSync_Rel[14]	:=	TRUE;
	bSync_Rel[15]	:=	TRUE;

	OUT_OP.tRel_Sync_Load.Do	:=	AND_Array(ADR(bSync_Rel),15);					(* 1 = sync is released *)
	OUT_OP.bRel_Sync_Load		:=	OUT_OP.tRel_Sync_Load.Do;
	MM2VIS.bSync_Rel			:=	bSync_Rel;						(* Array to VIS *)
	MM2VIS.bSync_Rel_Show		:=	(iIdx_Eng_State = 11) OR (iIdx_Eng_State = 12) OR (iIdx_Eng_State = 15) OR (iIdx_Eng_State = 16);

(** 39: State Machine *)
		(* MODULE BLOCKED *)
	IF 			OUT_OP.bEng_Bloc
		AND 	NOT bEng_StaSpdExc_old 			THEN
		iIdx_Eng_State := 19;

		(* ISLAND MODE - POWER MODE *)
	ELSIF 			IN_OP.tGCB_On.Di
		AND 		OUT_OP.tEng_Run.Do
		AND 	NOT IN_OP.tMCB_On.Di
		AND 	NOT IN_OP.bMCB_DemSy
		AND 		(IN_OP.bReq_PowMod OR IN_OP.bReq_PowMod_Ext)		THEN
		iIdx_Eng_State := 27;

		(* ISLAND MODE - SPEED MODE *)
	ELSIF 			IN_OP.tGCB_On.Di
		AND 		OUT_OP.tEng_Run.Do
		AND 	NOT	IN_OP.tMCB_On.Di
		AND 	NOT IN_OP.bMCB_DemSy
		AND 	NOT (IN_OP.bReq_PowMod OR IN_OP.bReq_PowMod_Ext)  	THEN
		iIdx_Eng_State := 26;

		(* EMERGENCY OPERATION *)		(* can never be used because AND FALSE !!! *)
	ELSIF 			IN_OP.tGCB_On.Di
		AND 		OUT_OP.tEng_Run.Do
		AND 		OUT_OP.bEng_Dem_EPS
		AND 	NOT IN_OP.bMCB_DemSy
		AND 		FALSE  						THEN
		iIdx_Eng_State := 18;

		(* PEAK LOAD OPERATION *)
	ELSIF 			IN_OP.tGCB_On.Di
		AND 		OUT_OP.tEng_Run.Do
		AND 	NOT	IN_OP.bMCB_DemSy
		AND 		IN_OP.tReq_PeakLoad.Di
		AND 		bOMSS_AUTO THEN
		iIdx_Eng_State := 23;

		(* GRID MODE *)
	ELSIF 			IN_OP.tGCB_On.Di
		AND 		OUT_OP.tEng_Run.Do
		AND 	NOT IN_OP.bMCB_DemSy 			THEN
		iIdx_Eng_State := 17;

		(* GRID MODE - WARM UP OPERATION *)
	ELSIF 			IN_OP.tGCB_On.Di
		AND 		OUT_OP.tEng_Run.Do
		AND 	NOT IN_OP.bMCB_DemSy
		AND			bWarmUpOperation	THEN
		iIdx_Eng_State := 37;

		(* BACK SYNCHRONIZATION *)
	ELSIF 			IN_OP.bMCB_DemSy
		AND 	NOT IN_OP.bBB_dead 		THEN
		iIdx_Eng_State := 16;

		(* SYNCHRONIZATION *)
	ELSIF 			IN_OP.bGCB_DemSy
		AND 	NOT IN_OP.bBB_dead 		THEN
		iIdx_Eng_State := 15;

		(* AFTER-COOLING *)
	ELSIF 			OUT_OP.bEng_CDR
		AND 	NOT OUT_OP.bEng_Dem_Man
		AND 	NOT OUT_OP.bEng_Dem_Aut
		AND 		OUT_OP.tEng_Run.Do 	THEN
		iIdx_Eng_State := 14;

		(* SHUT DOWN PHASE *)
	ELSIF 		(OUT_OP.bEng_Dem_Bloc OR OUT_OP.bEng_RSBoc OR IN_OP.bJmpPLTime)
		AND 	NOT OUT_OP.bEng_Dem_Man
		AND 	NOT OUT_OP.bEng_Dem_Aut
		AND  	NOT IN_OP.bSimWinMOD_FastStart		(* WinMOD *)
		AND 	NOT OUT_OP.tEng_Run.Do 	THEN
		iIdx_Eng_State := 13;	(* ABSTELLPHASE *)

		(* IDLE MODE / SY-LFG *)
	ELSIF 			OUT_OP.tRel_Sync_Load.Do
		AND 		OUT_OP.tEng_Run.Do 	THEN
		iIdx_Eng_State := 12;

		(* TEST *)
	ELSIF 			bOMSS_TEST
		AND 		OUT_OP.tEng_Run.Do 	THEN
		iIdx_Eng_State := 21;

		(* IDLE MODE / NO SY-LFG *)
	ELSIF 			OUT_OP.tEng_Run.Do 	THEN
		iIdx_Eng_State := 11;

		(* STANDBY TIME - AUTOMATIC START *)				(* Rev.4.03: new State 32: waiting for next automatic Start (for new BR4 start procedure)*)
	ELSIF 			(xTON_Eng_SU_Aut.Q OR (IN_OP.bSt_RelAuxOff_STT_op AND xEngType.Type6))   	 //	=delayed OUT_OP.bEng_SU_Aut  (Rev.4.04)
		AND 		OUT_OP.bEng_Dem_Aut
		AND 	NOT IN_OP.bEng_Start 	THEN
		iIdx_Eng_State := 32;

		(* prolonged normal start message *)				(* Rev.4.04: new State 33: demand automatic Start (for new BR4 start procedure)*)
	ELSIF 			OUT_OP.bEng_SU_Aut
		AND 		OUT_OP.bEng_Dem_Aut
		AND 	NOT IN_OP.bEng_Start 	THEN
		iIdx_Eng_State := 8;	(* Vorablösung: Wiederverwendung von 8=ENGINE START statt dem neuem iIdx_Eng_State := 33  prolonged normal start message;

		(* ENGINE START-UP *)
	ELSIF 			OUT_OP.bEng_Rel
		AND 	NOT OUT_OP.tEng_Run.Do
		AND 		IN_OP.bRelEngOp_Aux
		AND 	   (OUT_OP.bEng_Dem_Man OR OUT_OP.bEng_Dem_Aut)
		AND 		bEng_StaSpdExc
		AND 		IN_OP.bGV_On 		THEN
		iIdx_Eng_State := 10;

		(* AUTOMATIC START *)
	ELSIF 			OUT_OP.bEng_SU_Aut 	THEN
		iIdx_Eng_State := 9;

		(* ENGINE START *)
	ELSIF 			OUT_OP.bEng_Rel_SU
					AND NOT (OUT_OP.bEng_Dem_Man AND IN_OP.bSt_RelAuxOff_STT_op AND xEngType.Type6) 	THEN
		iIdx_Eng_State := 8;

		(* STANDBY TIME - MANUAL START *)
	ELSIF 			(OUT_OP.bEng_SU_Man
		AND 		OUT_OP.bEng_Dem_Man
		AND 	NOT OUT_OP.bEng_Rel_SU) OR
					(OUT_OP.bEng_Dem_Man AND IN_OP.bSt_RelAuxOff_STT_op AND xEngType.Type6) 	THEN
		iIdx_Eng_State := 7;

		(* PRELIMINARY PHASE *)
	ELSIF 			((OUT_OP.bEng_Aux_Dem AND OUT_OP.tEng_Aux_Dem_CDR.Do) OR IN_OP.bDemScavVa)
		AND 		(OUT_OP.bEng_Dem_Man OR OUT_OP.bEng_Dem_Aut)
		THEN
		iIdx_Eng_State := 6;

		(* TEST FINISHED *)
	ELSIF 			bOMSS_TEST
		AND 		OUT_OP.bEng_Rel 	THEN
		iIdx_Eng_State := 22;

		(* READY FOR AUTOMATIC VERY FAST START *)
	ELSIF 			OUT_OP.bEng_Rdy_Aut AND IN_OP.bReady4VeryFastStart	THEN
		iIdx_Eng_State := 33;

		(* READY FOR AUTOMATIC FAST START *)
	ELSIF 			OUT_OP.bEng_Rdy_Aut AND IN_OP.bReady4FastStart	THEN
		iIdx_Eng_State := 34;

		(* READY FOR AUTOMATIC START - VERY FAST START PREPERATION RUNNING *)
	ELSIF 			OUT_OP.bEng_Rdy_Aut AND IN_OP.bVeryFastStart_Prep	THEN
		iIdx_Eng_State := 35;

		(* READY FOR AUTOMATIC START - FAST START PREPERATION RUNNING *)
	ELSIF 			OUT_OP.bEng_Rdy_Aut AND IN_OP.bFastStart_Prep	THEN
		iIdx_Eng_State := 36;

		(* READY FOR AUTOMATIC FAST *)
	ELSIF 			OUT_OP.bEng_Rdy_Aut	THEN
		iIdx_Eng_State := 5;

		(* READY FOR MANUAL START *)
	ELSIF 			OUT_OP.bEng_Rdy_Man THEN
		iIdx_Eng_State := 4;

		(* OPERATION MODE SELECTOR SWITCH - TEST *)
	ELSIF 			bOMSS_TEST 		THEN
		iIdx_Eng_State := 20;

		(* OPERATION MODE SELECTOR SWITCH - AUTOMATIC *)
	ELSIF 			bOMSS_AUTO 		THEN
		iIdx_Eng_State := 3;

		(* OPERATION MODE SELECTOR SWITCH - MANUAL *)
	ELSIF 			bOMSS_MAN 		THEN
		iIdx_Eng_State := 2;

		(* OPERATION MODE SELECTOR SWITCH - OFF *)
	ELSIF 		NOT OUT_OP.tOMSS_MAT.Do		THEN
		iIdx_Eng_State := 1;

	END_IF;

(** 40: Engine operation hour counter *)
	(*This counter may be resetted in order to indicate an engine change*)
	xBH_OpHour(enable := OUT_OP.tEng_Run.Do, BH_adr := ADR(OpHour_Imp.tick));
	xTOF_OpHour(IN := xBH_OpHour.BH_Imp, PT := T#10s);
	OUT_OP.tImp_OpHour.Do :=  xTOF_OpHour.Q;

	IF EDGEPOS(IN_OP.iCnt_OpHours_Set > 0) AND bOpt_AllowCounterCorrection THEN		(*new in V4.13*)
			VIS2MM.iCnt_OpHours := IN_OP.iCnt_OpHours_Set;							(* Set counter intentionaly to database backup value from ParaBase module*)
	END_IF

	IF EDGEPOS(OUT_OP.tImp_OpHour.Do) THEN
		VIS2MM.iCnt_OpHours := DINT_INC_CNT(VIS2MM.iCnt_OpHours);						(* increase counter, check limits to +/- 1.000.000.000 *)
	END_IF
	OUT_OP.iCnt_OpHours := VIS2MM.iCnt_OpHours;

(** 41: Unit operation hour counter *)
	xBH_UnitOpHour(enable := OUT_OP.tEng_Run.Do, BH_adr := ADR(UnitOpHour_Imp.tick));
	xTOF_UnitOpHour(IN := xBH_UnitOpHour.BH_Imp, PT := T#10s);
	OUT_OP.bImp_UnitOpHour :=  xTOF_UnitOpHour.Q;

	IF EDGEPOS(IN_OP.iCnt_UnitOpHours_Set > 0) AND bOpt_AllowCounterCorrection THEN		(*new in V4.13*)
			VIS2MM.iCnt_UnitOpHours := IN_OP.iCnt_UnitOpHours_Set;						(* Set counter intentionaly to database backup value from ParaBase module*)
	END_IF

	IF EDGEPOS(OUT_OP.bImp_UnitOpHour) THEN
		VIS2MM.iCnt_UnitOpHours := DINT_INC_CNT(VIS2MM.iCnt_UnitOpHours);				(* increase counter, check limits to +/- 1.000.000.000 *)
	END_IF
	OUT_OP.iCnt_UnitOpHours := VIS2MM.iCnt_UnitOpHours;

(** 42: demand hour counter *)
	xBH_DemHour(enable := IN_OP.tDemEngOpExt.Di, BH_adr := ADR(DemHour_Imp.tick));
	xTOF_DemHour(IN := xBH_DemHour.BH_Imp, PT := T#10s);
	IF EDGEPOS(xTOF_DemHour.Q) THEN	(* if a demanded hour is finished *)
		VIS2MM.iCnt_DemHours := (VIS2MM.iCnt_DemHours + 1) MOD 1000000000;	(* increase counter, check limits *)
	END_IF;

(** 43: net parallel operation hour counter *)
	xBH_NetPHour(enable := xOpMode.NetP, BH_adr := ADR(NetPHour_Imp.tick));
	xTOF_NetPHour(IN := xBH_NetPHour.BH_Imp, PT := T#10s);
	IF EDGEPOS(xTOF_NetPHour.Q) THEN	(* if a mains operation hour is finished *)
		VIS2MM.iCnt_NetPHours := (VIS2MM.iCnt_NetPHours + 1) MOD 1000000000;	(* increase counter, check limits *)
	END_IF;

(** 44: island operation hour counter *)
	xBH_IslandHour(enable := xOpMode.Island, BH_adr := ADR(IslandHour_Imp.tick));
	xTOF_IslandHour(IN := xBH_IslandHour.BH_Imp, PT := T#10s);
	IF EDGEPOS(xTOF_IslandHour.Q) THEN	(* if an island operation hour is finished *)
		VIS2MM.iCnt_IslandHours := (VIS2MM.iCnt_IslandHours + 1) MOD 1000000000;	(* increase counter, check limits *)
	END_IF;

(** 45: start counter *)
	IF EDGEPOS(IN_OP.iCnt_Starts_Set > 0) AND bOpt_AllowCounterCorrection THEN		(*new in V4.13*)
			VIS2MM.iCnt_Starts := IN_OP.iCnt_Starts_Set;					(* Set counter intentionaly to database backup value from ParaBase module*)
	END_IF
	IF EDGEPOS(IN_OP.iCnt_FastStarts_Set > 0) AND bOpt_AllowCounterCorrection THEN	(*new in V4.13*)
			VIS2MM.iCnt_FastStarts := IN_OP.iCnt_FastStarts_Set;			(* Set counter intentionaly to database backup value from ParaBase module*)
	END_IF

	IF EDGEPOS(OUT_OP.bImp_Start) THEN
		VIS2MM.iCnt_Starts := DINT_INC_CNT(VIS2MM.iCnt_Starts);					(* increase counter, check limits to +/- 1.000.000.000 *)
		IF (IN_OP.iFastStart = 1) OR (IN_OP.iFastStart = 2) THEN
			VIS2MM.iCnt_FastStarts := DINT_INC_CNT(VIS2MM.iCnt_FastStarts);			(* increase counter, check limits to +/- 1.000.000.000 *)
		END_IF;
	END_IF;
	OUT_OP.iCnt_Starts 		:= VIS2MM.iCnt_Starts;
	OUT_OP.iCnt_FastStarts 	:= VIS2MM.iCnt_FastStarts;

(** 46: Low load operation counter *)
	xTON_OpLowLoadAct(IN := IN_OP.tGCB_On.Di, PT := T#5m);
 	bOpLowLoad := (OUT_OP.rP_Act_Norm_Filt < (Para.rP_Set_Min_Norm - 0.01)) AND xTON_OpLowLoadAct.Q AND M_ANF AND NOT IN_OP.bServiceMode;
	IF NOT bOpLowLoad THEN
		OpLowLoad_Imp.second := 0;
	END_IF;
	xBH_OpLowLoad(enable := bOpLowLoad, BH_adr := ADR(OpLowLoad_Imp.tick));
	xTOF_OpLowLoad(IN := xBH_OpLowLoad.BM_Imp, PT := T#10s);
	IF EDGEPOS(xTOF_OpLowLoad.Q) THEN
		VIS2MM.iCnt_OpLowLoad := DINT_INC_CNT(VIS2MM.iCnt_OpLowLoad);			(* increase counter, check limits to +/- 1.000.000.000 *)
	END_IF;

(** 47: logic war alarm 1108 and warning 2097 *)
	xTON_Rel_P_DevHi(IN:= OUT_OP.tEng_Run.Do AND bOMSS_AUTO AND IN_OP.tGCB_On.Di AND NOT OUT_OP.bEng_Dem_EPS, PT:= T#1200s);
	T99 := xTON_Rel_P_DevHi.Q;
	xGR_MAXR_P_Dev(In:= OUT_OP.rP_Set_Norm - OUT_OP.rP_Act_Norm_Filt, Gw:= Para.rP_Dev_LimHi, Hy:= 0.0);
	bP_DevHi := xGR_MAXR_P_Dev.Q AND IN_OP.tPB2MM.bParaSetupOk;
	xTON_P_DevHi(IN:= OUT_OP.bP_Rmp_Frz OR bP_DevHi, PT:= Para.tiP_Dev_LimHi_Delay);
	AN_PDIFF := xTON_P_DevHi.Q;

	UW_PDIFF_A := NOT xEngType.Type6 AND NOT xEngType.Type4 AND NOT Para.bEngTyp3_Prelub_Active;

(** 48: add submode to opstate status *)
	OUT_OP.iSt_OpMode := OUT_OP.iSt_OpMode OR 256 * iIdx_Eng_State;

(** 49: information operation mode for VISU *)
	xOpMode();
	iSt_OpMode_Main := xOpMode.iMainMode;
	iSt_OpMode_Sub := xOpMode.iSubMode;
	iSt_OpMode_Deg := xOpMode.iDegMode;

	bEng_StaSpdExc_old := bEng_StaSpdExc;

(** 50: new Out interfaces 4.7 *)
	(** 50.1: execute black out start, signal for customer *)
	IF EDGEPOS(OUT_OP.bEng_Dem_EPS) THEN
		OUT_OP.tExecute_BS.Do	:=	(NOT IN_OP.tAuxV_Eng_ok.Di AND IN_OP.tAuxV_Eng_ok.GoodQual)
								OR	(NOT IN_OP.tAuxV_Aux_ok.Di AND IN_OP.tAuxV_Aux_ok.GoodQual)
								OR	(NOT IN_OP.tAuxV_ModIf_ok.Di AND IN_OP.tAuxV_ModIf_ok.GoodQual)
								OR	(NOT IN_OP.tAuxV_Supply_Ok.Di AND IN_OP.tAuxV_Supply_Ok.GoodQual);
	END_IF
	IF xOpMode.Island OR xOpMode.NetP THEN
		OUT_OP.tExecute_BS.Do	:=	FALSE;
	END_IF

	OUT_OP.iIdx_Eng_State	:=	iIdx_Eng_State;

END_PROGRAM
```

#### op_state.fun
```iecst
(********************************************************************
 * COPYRIGHT -- INNIO Company
 ********************************************************************
 * Package: op_state
 * File: op_state.fun
 * Author: 502423184
 * Created: December 4, 2018
 *******************************************************************)

FUNCTION AND_Array : BOOL
	VAR_INPUT
		Adress : UDINT;
		Size : USINT;
	END_VAR
	VAR
		i : USINT;
		Arrayx : ARRAY[0..40] OF BOOL;
	END_VAR
END_FUNCTION

FUNCTION OR_Array : BOOL
	VAR_INPUT
		Adress : UDINT;
		Size : USINT;
	END_VAR
	VAR
		i : USINT;
		Arrayx : ARRAY[0..40] OF BOOL;
	END_VAR
END_FUNCTION

FUNCTION DINT_INC_CNT : DINT
	VAR_INPUT
		Input : DINT;
	END_VAR
END_FUNCTION
```

#### op_state.var
```iecst
VAR
	bPowerMode : BOOL;
	bEng_StaSpdExc_old : BOOL;
	ZM_H_ANF : BOOL;
	M_ABLOCK : BOOL;
	ZM_M_BERAUT : BOOL;
	bs_15s_rel_oper : BOOL;
	bs_15s_rpm_hi : BOOL;
	ZM_IN_bEng_CDR : BOOL;
	ZM_RS_bEng_CDR : BOOL;
	ZM_bEng_RSBoc : BOOL;
	xTON_RUN : TON;
	xTP_bEng_RSBoc : TP;
	xTOF_R_bEng_CDR : TOF_R;
	xTOF_SoftShutdown : TOF;
	xTON_T_Z_AUS : TON;
	xTP_AT27 : TP;
	xTON_T105 : TON;
	xTOF_ANFBLO : TOF;
	xTOF_T9 : TOF;
	xTOF_Eng_Aux_Dem : TOF;
	xTON_kwtp : TON;
	xTOF_Eng_StaSpdExc : TOF;
	xTP_Imp_Start : TP;
	xTOF_BlocDelay_ManStart : TOF; (*Pulse generator for engine start*)
	xGR_MAXR_Eng_StaSpdExc : GR_MAXR;
	xGR_MAXR_bs_15s_rpm_hi : GR_MAXR;
	xGRMinR_KWT : GR_MINR;
	xBH_UnitOpHour : BH; (*Unit operating hours counter*)
	xTOF_UnitOpHour : TOF; (*10 seconds delay for engine begin of operation*)
	xBH_OpHour : BH; (*Hour counter for engine operating hours*)
	xTOF_OpHour : TOF; (*Off delay for engine operating hours*)
	xGR_MINR_P_Lo : GR_MINR;
	xTON_Rel_P_DevHi : TON;
	xGR_MAXR_P_Dev : GR_MAXR;
	xTON_P_DevHi : TON;
	xGR_MAXR_OpenGV : GR_MAXR;
	xTP_OpenGV : TP;
	bStop2Start : BOOL; (*transition from stop state to start state*)
	bRSS_OFF : BOOL;
	bRSS_ON : BOOL;
	bIgn_DemTemp : BOOL; (*Wegen Abstellstörung 1023 und Auftreten von 1056*)
	Ign_Dem_DelayTime : TIME := T#200ms; (*Wegen Abstellstörung 1023 und Auftreten von 1056*)
	xTOFIgn_Dem : TOF; (*Wegen Abstellstörung 1023 und Auftreten von 1056*)
	xTOF_OFF : TOF;
	xTOF_MAN : TOF;
	xTOF_AUTO : TOF;
	xTOF_TEST : TOF;
	xTOF_SCAV : TOF;
	xTON_Eng_SU_Aut : TON; (*new for V4.04 - State 32*)
	xBH_DemHour : BH; (*Engine demand hours counter*)
	xTOF_DemHour : TOF; (*Off delay for engine demand*)
	xBH_NetPHour : BH; (*Engine grid running hours counter*)
	xTOF_NetPHour : TOF; (*Off delay for engine grid running*)
	xBH_IslandHour : BH; (*Engine island running hours counter*)
	xTOF_IslandHour : TOF; (*Off delay for engine island running*)
	IslandHour_Imp : bh_typ; (* Island Operation Hour Counter*)
	NetPHour_Imp : bh_typ; (* Net Parallel Operation Hour Counter*)
	DemHour_Imp : bh_typ; (* Demand Hour Counter*)
	rN_Eng_Limit : REAL := 1545; (* Speed Limit for type 6 housload rejection [rpm] *)
	bTrigger_Island : BOOL; (* island trigger for type 6 housload rejection *)
	tOff_Trigger : TIME := T#1s; (* Duration island trigger for type 6 housload rejection *)
	TOF_bTrigger_Island : TOF;
	bDryTestBench : BOOL := 0; (*DONT TOUCH THIS SIGNAL!*)
	bEng_Bloc : ARRAY[0..50] OF BOOL;
	bSync_Rel : ARRAY[0..15] OF BOOL;
	bEng_SU : ARRAY[0..6] OF BOOL;
	bIgn_Dem : ARRAY[0..5] OF BOOL;
	bEng_Dem_A : ARRAY[0..9] OF BOOL;
	bRequest_A : BOOL;
	bRequest_EPS : BOOL := 0;
	bGV_Open : ARRAY[0..7] OF BOOL;
	bReq_Dem : ARRAY[0..7] OF BOOL;
	bRequest_Dem : BOOL;
	bReq_Bloc : ARRAY[0..6] OF BOOL;
	bReq_A : ARRAY[0..5] OF BOOL;
	bT_ECW_Lo : BOOL; (* AN_KTMI wird lokal gebildet und nur im modul verwendet *)
	bN_Eng_Run : BOOL; (*Speed Condition ok for Eng_Run*)
	xTON_Block_PlantCtr : TON;
	TOF_b2973 : TOF;
	xTOF_EngDemEPS : TOF;
	Ign_Dem_DelayTime2 : TIME := T#200ms;
	bOpt_AllowCounterCorrection : BOOL := TRUE; (*Allways TRUE, except for debugging*)
	xBH_OpLowLoad : BH; (* Low load operation counter *)
	OpLowLoad_Imp : bh_typ; (* Low load operation minutes counter*)
	xTON_OpLowLoadAct : TON; (* Delay after GCB-On for low load operation counter *)
	bOpLowLoad : BOOL; (* Low load operation counter active *)
	xTOF_OpLowLoad : TOF; (* Ten second pulse for low load operation counter *)
END_VAR
```

### Program Logical/Opstate/powersel (IEC) - + Power Setpoint selection

- powerselCyclic.st (not readable text: treated as protected, skipped)

- powerselInit.st (not readable text: treated as protected, skipped)

#### powersel.var
```iecst
VAR
	rP_Set_Min_Norm : REAL; (*Minimum power setpoin p.u.*)
	rP_Set_Norm : REAL;
	bRampEnable : BOOL; (* TRUE=setpoint power ramp active *)
	xRAMPE_SetPower : LCRRamp;
	bLastNetpM : BOOL;
	bLeftInsel : BOOL;
	i : USINT;
	rP_Nom_Gastype : REAL;
	rP_Ramp_IncGrad_Norm : REAL;
	rP_Ramp_DecGrad_Norm : REAL;
	TP_GasMixing : TP;
	iIdx_Gtyp_Dem_old : INT;
	bGasMixingActive_old : BOOL;
	bGEN2FastRamp : BOOL;
	rP_Set_Max_Norm : REAL;
	do_Nothing : BOOL;
	bPRed_Loop : BOOL;
	iIdx_Pset_Type : INT; (* power setpoint: 1 = VIS, 2 = AI, 3 = BUS, 4 = CUST, 5 = PFC, 6 = EU, 7 = Mns, 8 = PU, 9 = WUO *)
	TON_ParaSetupOk_2s : TON;
	bAct_CompMGC_Nfilter : BOOL := TRUE;
	xLCRPT1_Nact : LCRPT1; (*Compatibility to Microgrid Ctrl: Speed Filter*)
	rN_EngAct_filt : REAL := 1500;
	rP_offs_CompMGC_1 : REAL := 0.0;
	rP_offs_CompMGC_2 : REAL := 0.0;
	rP_offs_CompMGC_2upd : REAL := 0.0;
	bTest_CompMGC_extNoffset : BOOL;
	rN_Offs_Cust : REAL := 0.00;
	rK_CompMGC_extNoffset : REAL := 0.001; (* Compatibility to Microgrid Ctrl: scaling factor *)
	dN : REAL := 0.0;
	rNdiff_Lim_CompMGC : REAL := 90.0;
	bSyDemand : BOOL := 0;
	tTof_ActCompMGC_Sy : TIME := T#1s;
	xTOF_SyDemand : TOF;
	rP_offs_CompMGC_2_max : REAL;
	rP_DiffMax_CompMGC_2 : REAL := 0.05;
	rP_offs_CompMGC_2_min : REAL;
	R_TRIG_Event_Change  : R_TRIG; (* Trigger bit for event change in case of power set point via bus *)
END_VAR
```

### Program Logical/Opstate/speedsel (IEC) - + Speed Selection

- speedselCyclic.st (not readable text: treated as protected, skipped)

- speedselInit.st (not readable text: treated as protected, skipped)

#### speedsel.var
```iecst
VAR
	rN_Sync_Delta_Norm : REAL := 0.0;
	bInitRamp : BOOL;
	xLCRRAMP_IslandLoading : LCRRamp;
	xLCRRAMP_N_Delta : LCRRamp;
	rN_Loadsharing_Delta_Norm : REAL := 0.0;
	rLoadsharing_Scal : REAL := 0.1; (*control gain for engine speed set value of load sharing line*)
	DEM_ISOL : BOOL;
	anz_vmod : REAL;
	wert1 : REAL;
	wert2 : REAL;
	wert3 : REAL;
	wert4 : REAL;
	wert_unten : REAL;
	wert_oben : REAL;
	xRamp_GH_lsl : RAMPE_R;
	rCnt_Pmax : REAL;
	bPDrift_Rel : BOOL;
	bPDrift_Ena : BOOL;
	rP_Avg_Norm : REAL;
	rP_Set_ext_Norm : REAL;
	rP_Dev_Norm : REAL;
	rP_Dev_Lim : REAL;
	rP_Offs : REAL;
	rF_Offs : REAL;
	rP_Max : REAL;
	rP_Offs_Input : REAL;
	xRAMPE_R_Droop : RAMPE_R;
	rF_Offs_Norm : REAL;
	xLCRScal_F_WPt : LCRScal := (0);
	x_win : ARRAY[0..1] OF REAL;
	xLCRRamp_N_Set_Offset : LCRRamp;
	rN_F_Offset : REAL;
	rP_Red_Norm_Island_Set : REAL;
	xFILTER_R_P_Act_Norm : FILTER_R;
	rN_F_Offset_Old : REAL;
	rP_Offs_Input_0kW : REAL;
	rN_Offs_notDem : REAL := 10; (* [rpm] offset if engine not demanded, in external speed reference mode*)
	rP_OffsInit : REAL := 0.0;
	bAddDroop_NrefExt : BOOL := TRUE; (* activate additional droop fro external speed ref.*)
	rN_F_Offset_AddDroop : REAL := 0.0; (* additional droop term for external speed ref. *)
	rLim_AddDroop : REAL := 1; (* Limit for additional droop *)
	rN_delta_OvldProt : REAL; (*Spd Ctrl, speed ref. offset for overload protection *)
	bDroopPowCtrl : BOOL; (*Compatibility to Microgrid Ctrl: droop for power controller active*)
	rN_delta_RevPowProt : REAL := 0.0; (*Spd Ctrl, speed ref. offset for reverse power protection*)
	xLCRPT1_PActNorm_LoadProt : LCRPT1; (*Filter of actual power for load protection*)
	rN_F_Offset_norm_lim : REAL := 0.06; (*normalized speed ref. offset limit*)
	xRAMPE_R_overLoadProt : RAMPE_R := (0); (*rate limiter for output of the overload protection*)
	xRAMPE_R_reversePowerProt : RAMPE_R := (0); (*rate limiter for output of the reverse power protection*)
	rN_Gradient_Ramps_LoadProtection : REAL := 0.0; (*gradient of load protection rate limiter *)
	rN_delta_OvldProt_Cont : REAL := 0.0; (*speed offset from overload protection p controller*)
	rN_delta_RevPowProt_Cont : REAL := 0.0; (*speed offset from reverse power protection p controller*)
	rFact_Rampback_Loadprotection : REAL; (*Factor for ramp gradient ramping back from overload or reverse power reaction*)
	xR_Trig_LSLTransition : R_TRIG; (*rising edge trigger used for LSL transitions *)
	bOtherGensInLSL : BOOL; (*TRUE if other generators in parallel participating in the LSL *)
	rP_Island_Split_Max : REAL; (*Maximum of the rP_Island_Split variable *)
	xLCRRamp_LSLTransition : LCRRamp; (*Ramp used for smooth transition to LSL *)
	rN_Grad_LSLTransition : REAL; (*Gradient used for smooth transition to LSL *)
	xLCRIntegrate_LSL_Correction : LCRIntegrate; (*Integrator for LSL signal error compensation *)
END_VAR
```

### Program Logical/Opstate/MsgOP (IEC) - OpState Messages

#### MsgOPCyclic.st - OpState Messages Cyclic
```iecst
(*******************************************************************************
MsgOG	 			 alarms generation MM_Opstate

This code is confidential and proprietary to the INNIO Company.
It may not be used in any form, or reproduced in any manner,
without written permission of the INNIO Company.
Copyright, INNIO Company, 2023

Customized modifications: -
------------------------

History:
-------
V3.99.0	xx-03-2012	Graus		new
		27.05.2013	Lettenb.	reset OUT_xx.txx2AB.bGnlTripx changed
		05.10.2013	Graus,		add messages bMsg2122, bMsg2123, bMsg2124
V4.00.0 11.02.2014 	Graus,		change Version TO 4.0
		04.03.2014	lettenb.	logger added
V4.01.0	18.07.2014	Graus,		use both staticGR power reductions for same operation message (bP_Red_EVU OR bP_Red_EU)
V4.04.0 11.02.2014 	Graus,		change Version TO 4.04
V4.04.0 17.11.2016	Gomez Ortiz	Addition of B2168 generator air inlet temperature power reduction
V4.05.0 14.06.2017	Gomez Ortiz Addition OF power limitation due TO low engine cooling water temperature, Spec_Start_Load_release_manual_start.doc
V4.05.1	25.09.2017  Gomez Ortiz Removal of UW_PDIFF_A (engine type dependency) from the Alarm 1108 and Alarm 2097
V4.05.2	24.10.2017	Zingerle	SWAT 920 Rel.5, power reduction with difference pressure minimum (bMsg2936)
V4.07.0	11.07.2018	Messner,	CPP Integrator - B2961 added
		23.10.2018	Maran,		implemented B2983 - B2985 for request selector switch positions
V4.07.4	29.03.2019	Hohensinner	Bugfixing: added W9284
V4.07.5	15.05.2019	Hohensinner	added EngBlock_PlantCtr DI to W1188
V4.09.0 03.02.2020	Zuschnig	included TOF (60s) for operation message B1283 to B1287
		12.02.2020	Zuschnig	included B2972 and B2973 - Power Mode on/off and ParaSetupOk plus 2 sec for B2140
V4.11.0	23.04.2021  Zuschnig	Bugfix - B2154 triggered with high frequency bit
        20.08.2021 	Keller		Add Messages 9051, 9052, 9061, 9062
		22.11.2021	Perktold,	added B9063, B9064
		22.12.2021	Andre		added B2935 Power reduction by CAN communication failure for half or more SAFI or too many SAFI reboots
		01.04.2022	Zuschnig 	TOF with 60s for messages 2130, 2152, 2153 and 2154 to prevent too many messages
V4.12.0	12.01.2023  Tinello		Deleted power reduction by T1HP (2803) / Added power reduction by T2HP (9075) and T2LP (9076)
    	16.01.2023  Zuschnig	TOF with 60s for message 2989 to prevent too many messages
		22.01.2023  Zuschnig	Include B9072 - Power reduction by H2 content

Instructions for use:
--------------------
1) declare alarm with function block "Alm"
	declare buffert alarm bit bMsg<message number>

2) use template to create a new alarm,
   substitue 0000 by alarm number and make settings:

	xMsg0000.Enable		:=	TRUE;		enable/disable alarm
	xMsg0000.Set		:=	FALSE;		alarm set condition
	xMsg0000.PT			:=	T#0s;		alarm delay time
	xMsg0000.Prio		:=	1;			alarm priority: 1-3 = trip, 4 = warning
	xMsg0000.RiskClass	:=	3;			risk class for remote alarm reset
	xMsg0000.Reset		:=	FALSE;		FALSE: for all standard alarms	prio 1,2,3 and warnings prio 4
										TRUE : for autoreset alarms

	bMsg0000			:=	xMsg0000.Q;	connect buffert alarm bit for VIS and control

3)  expand INIT

3)	include datapoint into OPC configuration for vis

Outstandings:
------------
(*******************************************************************************)
PROGRAM _CYCLIC

	(* reset general trip *)
	OUT_OP.tOP2AB.bGnlTrip1			:=	FALSE;
	OUT_OP.tOP2AB.bGnlTrip2			:=	FALSE;
	OUT_OP.tOP2AB.bGnlTrip3			:=	FALSE;
	OUT_OP.tOP2AB.bGnlWarning		:=	FALSE;
	OUT_OP.tOP2AB.bTriptype1		:=	FALSE;
	OUT_OP.tOP2AB.bTriptype2		:=	FALSE;
	OUT_OP.tOP2AB.bTriptype3		:=	FALSE;

	(*---------------------------------------------------------------------------*)
	// Alarms and warnings

	(* A1108 actual power deviation maximum *)
	xMsg1108.Enable		:=	FALSE;
	xMsg1108.Set		:=	AN_PDIFF AND T99;			(*Gomez Ortiz, no more engine type dependency for this alarm setting*)
	xMsg1108.PT			:=	T#0s;
	xMsg1108.Prio		:=	3;
	xMsg1108.RiskClass	:=	4;
	xMsg1108.Reset		:=	FALSE;
	xMsg1108();
	bMsg1108			:= xMsg1108.Q;
	OUT_OP.bMsg1108 	:= xMsg1108.Q;

	(* W3506 Power reduction in isolated operation *)
	xMsg3506.Enable		:=	TRUE;
	xMsg3506.Set		:=	bPRed_Active AND xOpMode.Island;
	xMsg3506.PT			:=	T#0s;
	xMsg3506.Prio		:=	4;
	xMsg3506.RiskClass	:=	4;
	xMsg3506.Reset		:=	FALSE;
	xMsg3506();
	bMsg3506			:= xMsg3506.Q;

	(* W2082 Warning: Parameters missing *)
	xMsg2082.Enable		:=	TRUE;
	xMsg2082.Set		:=	RPSW_1;
	xMsg2082.PT			:=	T#0s;
	xMsg2082.Prio		:=	4;
	xMsg2082.RiskClass	:=	4;
	xMsg2082.Reset		:=	FALSE;
	xMsg2082();
	bMsg2082			:= xMsg2082.Q;

	(* W1188 release by station missing *)
	xMsg1188.Enable		:=	TRUE;
	xMsg1188.Set		:=	NOT AT27 OR bEng_Block_PlantCtr;
	xMsg1188.PT			:=	T#0s;
	xMsg1188.Prio		:=	4;
	xMsg1188.RiskClass	:=	4;
	xMsg1188.Reset		:=	IN_OP.tEngBlock_PlantCtr.GoodQual;
	xMsg1188();
	bMsg1188			:= xMsg1188.Q;

	(* W2097 Leistungsistwertabweichung Maximum *)
	xMsg2097.Enable		:=	TRUE;
	xMsg2097.Set		:=	AN_PDIFF AND T99;	(*Gomez Ortiz, no more engine type dependency for this alarm setting*)
	xMsg2097.PT			:=	T#0s;
	xMsg2097.Prio		:=	4;
	xMsg2097.RiskClass	:=	4;
	xMsg2097.Reset		:=	FALSE;
	xMsg2097();
	bMsg2097			:= xMsg2097.Q;

	(* W9284 Measuring signal failure External power set point for Speed droop mode *)
	xMsg9284.Enable		:=	IN_OP.tPB2MM.bParaSetupOk AND IN_OP.tP_Droop_Set.Exist AND (IN_OP.iSource_F_N_OffsSet = 1);
	xMsg9284.Set		:=	NOT IN_OP.tP_Droop_Set.GoodQual;
	xMsg9284.PT			:=	T#1s;
	xMsg9284.Prio		:=	4;
	xMsg9284.RiskClass	:=	4;
	xMsg9284.Reset		:=	FALSE;
	xMsg9284();
	MM2VIS.bMsg9284		:= xMsg9284.Q;

	(*-----------------------------------------------------------------------*)
	(* operating messages > AMM *)

	(* B2125 P reduction by knocking (diagn.msg RPS) *)
	xMsg2125.Enable		:=	TRUE;
	xMsg2125.Set		:=	xPRed[_Knck].Q;
	xMsg2125.Reset		:=	TRUE;
	xMsg2125();
	bMsg2125			:=	xMsg2125.Q;

	(* B2126 P reduction by mixture temp. (diagn.msg RPS) *)
	xMsg2126.Enable		:=	TRUE;
	xMsg2126.Set		:=	xPRed[_TMix].Q AND IN_OP.tGCB_On.Di;
	xMsg2126.Reset		:=	TRUE;
	xMsg2126();
	bMsg2126			:=	xMsg2126.Q;

	(* B2127 P reduction by misfiring (diagn.msg RPS) *)
	xMsg2127.Enable		:=	TRUE;
	xMsg2127.Set		:=	xPRed[_Misf].Q;
	xMsg2127.Reset		:=	TRUE;
	xMsg2127();
	bMsg2127			:=	xMsg2127.Q;

	(* B2128 P reduction by external(analoge) (diagn.msg RPS) *)
	xMsg2128.Enable		:=	TRUE;
	xMsg2128.Set		:=	xPRed[_AI].Q;
	xMsg2128.Reset		:=	TRUE;
	xMsg2128();
	bMsg2128			:=	xMsg2128.Q;

	(* B2129 P reduction by external(bus) (diagn.msg RPS) *)
	xMsg2129.Enable		:=	TRUE;
	xMsg2129.Set		:=	xPRed[_EBus].Q;
	xMsg2129.Reset		:=	TRUE;
	xMsg2129();
	bMsg2129			:=	xMsg2129.Q;

	(* B2130 P reduction by frequency low (diagn.msg RPS) *)
	xTOF_Msg2130(IN:= xPRed[_F_Lo].Q, PT := T#60s);

	xMsg2130.Enable		:=	TRUE;
	xMsg2130.Set		:=	xTOF_Msg2130.Q;
	xMsg2130.Reset		:=	TRUE;
	xMsg2130();
	bMsg2130			:=	xMsg2130.Q;

	(* B2131 maximum output limit *)
	xMsg2131.Enable		:=	TRUE;
	xMsg2131.Set		:=	xPRed[_PMax].Q;
	xMsg2131.Reset		:=	TRUE;
	xMsg2131();
	bMsg2131			:=	xMsg2131.Q;

	(* B2132 P reduction by cyl.temp. (diagn.msg RPS) *)
	xMsg2132.Enable		:=	TRUE;
	xMsg2132.Set		:=	xPRed[_EGT].Q;
	xMsg2132.Reset		:=	TRUE;
	xMsg2132();
	bMsg2132			:=	xMsg2132.Q;

	(* B2140 demand for island operation *)
	xMsg2140.Enable		:=	TRUE;
	xMsg2140.Set		:=	OUT_OP.bEng_Dem_EPS AND NOT IN_OP.bOnly_Island AND bParaSetupOk_2s;(* M_NANF AND NOT REIN_INSEL *)
	xMsg2140.Reset		:=	TRUE;
	xMsg2140();
	bMsg2140			:=	xMsg2140.Q;

	(*B2143 P reduction by air intake temp. (diagn.msg RPS) *)
	xMsg2143.Enable		:=	TRUE;
	xMsg2143.Set		:=	xPRed[_T1LP].Q;
	xMsg2143.Reset		:=	TRUE;
	xMsg2143();
	bMsg2143			:=	xMsg2143.Q;

	(* B2144 P reduction by turbo charger speed high (diagn.msg RPS) *)
	xMsg2144.Enable		:=	TRUE;
	xMsg2144.Set		:=	xPRed[_N_TC].Q;
	xMsg2144.Reset		:=	TRUE;
	xMsg2144();
	bMsg2144			:=	xMsg2144.Q;

	(* B2146 PBC power reduction *)
	xMsg2146.Enable		:=	TRUE;
	xMsg2146.Set		:=	xPRed[_PBC].Q;
	xMsg2146.Reset		:=	TRUE;
	xMsg2146();
	bMsg2146			:=	xMsg2146.Q;

	(* B2147 P reduction by leanox ctrl.deviation high (diagn.msg RPS) *)
	xMsg2147.Enable		:=	TRUE;
	xMsg2147.Set		:=	xPRed[_LX].Q;
	xMsg2147.Reset		:=	TRUE;
	xMsg2147();
	bMsg2147			:=	xMsg2147.Q;

	(* B2148 diagn.msg RPS 28 *)
	xMsg2148.Enable		:=	TRUE;
	xMsg2148.Set		:=	xPRed[_SP1].Q;
	xMsg2148.Reset		:=	TRUE;
	xMsg2148();
	bMsg2148			:=	xMsg2148.Q;

	(* B2149 diagn.msg RPS 29 *)
	xMsg2149.Enable		:=	TRUE;
	xMsg2149.Set		:=	xPRed[_SP2].Q;
	xMsg2149.Reset		:=	TRUE;
	xMsg2149();
	bMsg2149			:=	xMsg2149.Q;

	(* B2150 diagn.msg RPS 30 *)
	xMsg2150.Enable		:=	TRUE;
	xMsg2150.Set		:=	xPRed[_SP3].Q;
	xMsg2150.Reset		:=	TRUE;
	xMsg2150();
	bMsg2150			:=	xMsg2150.Q;

	(* B2152 P reduction by voltage low  (diagn.msg RPS) *)
	xTOF_Msg2152(IN:= xPRed[_U_Lo].Q, PT := T#60s);

	xMsg2152.Enable		:=	TRUE;
	xMsg2152.Set		:=	xTOF_Msg2152.Q;
	xMsg2152.Reset		:=	TRUE;
	xMsg2152();
	bMsg2152			:=	xMsg2152.Q;

	(* B2153 P reduction by voltage high (diagn.msg RPS) *)
	xTOF_Msg2153(IN:= xPRed[_U_Hi].Q, PT := T#60s);

	xMsg2153.Enable		:=	TRUE;
	xMsg2153.Set		:=	xTOF_Msg2153.Q;
	xMsg2153.Reset		:=	TRUE;
	xMsg2153();
	bMsg2153			:=	xMsg2153.Q;

	(* B2154 P reduction by frequency high (diagn.msg RPS) *)
	xTOF_Msg2154(IN:= xPRed[_F_Hi].Q, PT := T#60s);

	xMsg2154.Enable		:=	TRUE;
	xMsg2154.Set		:=	xTOF_Msg2154.Q;
	xMsg2154.Reset		:=	TRUE;
	xMsg2154();
	bMsg2154			:=	xMsg2154.Q;

	(* B2155 P reduction by gen.winding temp. (diagn.msg RPS) *)
	xMsg2155.Enable		:=	TRUE;
	xMsg2155.Set		:=	xPRed[_GWT].Q;
	xMsg2155.Reset		:=	TRUE;
	xMsg2155();
	bMsg2155			:=	xMsg2155.Q;

	(* B2158 P reduction by jacket water temperature (diagn.msg RPS) *)
	xMsg2158.Enable		:=	TRUE;
	xMsg2158.Set		:=	xPRed[_JWT].Q;
	xMsg2158.Reset		:=	TRUE;
	xMsg2158();
	bMsg2158			:=	xMsg2158.Q;

	(* B2159 P reduction by oil temperature (diagn.msg RPS) *)
	xMsg2159.Enable		:=	TRUE;
	xMsg2159.Set		:=	xPRed[_OILT].Q;
	xMsg2159.Reset		:=	TRUE;
	xMsg2159();
	bMsg2159			:=	xMsg2159.Q;

	(* B2160 P reduction by heating water return temperature (diagn.msg RPS) *)
	xMsg2160.Enable		:=	TRUE;
	xMsg2160.Set		:=	xPRed[_RWT].Q;
	xMsg2160.Reset		:=	TRUE;
	xMsg2160();
	bMsg2160			:=	xMsg2160.Q;

	(* B2161 P reduction by pressure pre chamber gas train (diagn.msg RPS) *)
	xMsg2161.Enable		:=	TRUE;
	xMsg2161.Set		:=	xPRed[_PCGT].Q;
	xMsg2161.Reset		:=	TRUE;
	xMsg2161();
	bMsg2161			:=	xMsg2161.Q;

	(* B2163 Power reduction by utility *)
	xMsg2163.Enable		:=	TRUE;
	xMsg2163.Set		:=	xPRed[_EVU].Q OR xPRed[_EU].Q;
	xMsg2163.Reset		:=	TRUE;
	xMsg2163();
	bMsg2163			:=	xMsg2163.Q;

	(* B2164 Power limitation by air humidity *)
	xMsg2164.Enable		:=	TRUE;
	xMsg2164.Set		:=	xPRed[_Hum].Q;
	xMsg2164.Reset		:=	TRUE;
	xMsg2164();
	bMsg2164			:=	xMsg2164.Q;

	(* B2170 power redutcion by hierarchy controller *)
	xMsg2170.Enable		:=	TRUE;
	xMsg2170.Set		:=	xPRed[_HiCtr].Q;
	xMsg2170.Reset		:=	TRUE;
	xMsg2170();
	bMsg2170			:=	xMsg2170.Q;

	(* B2169 power redutcion by  timing point optimizing *)
	xMsg2169.Enable		:=	TRUE;
	xMsg2169.Set		:=	xPRed[_IPOpt].Q;
	xMsg2169.Reset		:=	TRUE;
	xMsg2169();
	bMsg2169			:=	xMsg2169.Q;

	(* B2803 power reduction by charge temp.before HP TC *)			(* --> NOT USED >= v4.12 *)
	xMsg2803.Enable		:=	FALSE;
	xMsg2803.Set		:=	FALSE;
	xMsg2803.Reset		:=	TRUE;
	xMsg2803();
	bMsg2803			:=	xMsg2803.Q;

	(* B2936 Power reduction by pressure gas train min  *)
	xMsg2936.Enable		:=	TRUE;
	xMsg2936.Set		:=	xPRed[_PrGR].Q;
	xMsg2936.Reset		:=	TRUE;
	xMsg2936();
	bMsg2936			:=	xMsg2936.Q;

	(* B3229 P reduction by CH4 content  (diagn.msg RPS) *)
	xMsg3229.Enable		:=	TRUE;
	xMsg3229.Set		:=	xPRed[_CH4].Q;
	xMsg3229.Reset		:=	TRUE;
	xMsg3229();
	bMsg3229			:=	xMsg3229.Q;

	(* B3230 P reduction by gas pressure (diagn.msg RPS) *)
	xMsg3230.Enable		:=	TRUE;
	xMsg3230.Set		:=	xPRed[_GasPr].Q;
	xMsg3230.Reset		:=	TRUE;
	xMsg3230();
	bMsg3230			:=	xMsg3230.Q;

	(* B3231 P reduction by suction pressure (diagn.msg RPS) *)
	xMsg3231.Enable		:=	TRUE;
	xMsg3231.Set		:=	xPRed[_Suct].Q;
	xMsg3231.Reset		:=	TRUE;
	xMsg3231();
	bMsg3231			:=	xMsg3231.Q;

	(* op_msg *)

	(* B1225 service seletion switch off *)
	xMsg1225.Enable		:=	TRUE;
	xMsg1225.Set		:=	(OUT_OP.iIdx_OMSS = 0);
	xMsg1225.Reset		:=	TRUE;
	xMsg1225();
	bMsg1225			:=	xMsg1225.Q;

	(* B1226 service seletion switch manual *)
	xMsg1226.Enable		:=	TRUE;
	xMsg1226.Set		:=	(OUT_OP.iIdx_OMSS = 1);
	xMsg1226.Reset		:=	TRUE;
	xMsg1226();
	bMsg1226			:=	xMsg1226.Q;

	(*B1227 service seletion switch automatic *)
	xMsg1227.Enable		:=	TRUE;
	xMsg1227.Set		:=	(OUT_OP.iIdx_OMSS = 2);
	xMsg1227.Reset		:=	TRUE;
	xMsg1227();
	bMsg1227			:=	xMsg1227.Q;

	(* B1228 service seletion switch test *)
	xMsg1228.Enable		:=	TRUE;
	xMsg1228.Set		:=	(OUT_OP.iIdx_OMSS = 3);
	xMsg1228.Reset		:=	TRUE;
	xMsg1228();
	bMsg1228			:=	xMsg1228.Q;

	(* B1229 engine ready for automatic on  *)
	xMsg1229.Enable		:=	TRUE;
	xMsg1229.Set		:=	OUT_OP.bEng_Rdy_Aut;
	xMsg1229.Reset		:=	TRUE;
	xMsg1229();
	bMsg1229			:=	xMsg1229.Q;

	(* B1230 engine ready for automatic off *)
	xMsg1230.Enable		:=	TRUE;
	xMsg1230.Set		:=	NOT	OUT_OP.bEng_Rdy_Aut;
	xMsg1230.Reset		:=	TRUE;
	xMsg1230();
	bMsg1230			:=	xMsg1230.Q;

	(* B1231 engine demand on  *)
	xMsg1231.Enable		:=	TRUE;
	xMsg1231.Set		:=	OUT_OP.bEng_Dem;
	xMsg1231.Reset		:=	TRUE;
	xMsg1231();
	bMsg1231			:=	xMsg1231.Q;

	(* B1232 engine demand off *)
	xMsg1232.Enable		:=	TRUE;
	xMsg1232.Set		:=	NOT OUT_OP.bEng_Dem;
	xMsg1232.Reset		:=	TRUE;
	xMsg1232();
	bMsg1232			:=	xMsg1232.Q;

	(* B1233 engine operation on  *)
	xMsg1233.Enable		:=	TRUE;
	xMsg1233.Set		:=	OUT_OP.tEng_Run.Do;
	xMsg1233.Reset		:=	TRUE;
	xMsg1233();
	bMsg1233			:=	xMsg1233.Q;

	(* B1234 engine operation off *)
	xMsg1234.Enable		:=	TRUE;
	xMsg1234.Set		:=	NOT OUT_OP.tEng_Run.Do;
	xMsg1234.Reset		:=	TRUE;
	xMsg1234();
	bMsg1234			:=	xMsg1234.Q;

	(* B1237 demand for island operation on  *)
	xMsg1237.Enable		:=	TRUE;
	xMsg1237.Set		:=	OUT_OP.bEng_Dem_EPS AND FALSE;
	xMsg1237.Reset		:=	TRUE;
	xMsg1237();
	bMsg1237			:=	xMsg1237.Q;

	(* B1238 demand for island operation off *)
	xMsg1238.Enable		:=	TRUE;
	xMsg1238.Set		:=	NOT OUT_OP.bEng_Dem_EPS AND FALSE;
	xMsg1238.Reset		:=	TRUE;
	xMsg1238();
	bMsg1238			:=	xMsg1238.Q;

	(* B1241 selection gas type 1  *)
	xMsg1241.Enable		:=	TRUE;
	xMsg1241.Set		:=	OUT_OP.bGasTyp1_Act AND (IN_OP.iIdx_Gtyp_Dem = 1);
	xMsg1241.Reset		:=	TRUE;
	xMsg1241();
	bMsg1241			:=	xMsg1241.Q;

	(* B1242 selection gas type 2  *)
	xMsg1242.Enable		:=	TRUE;
	xMsg1242.Set		:=	OUT_OP.bGasTyp2_Act;
	xMsg1242.Reset		:=	TRUE;
	xMsg1242();
	bMsg1242			:=	xMsg1242.Q;

	(*  B1243 selection gas type 3  *)
	xMsg1243.Enable		:=	TRUE;
	xMsg1243.Set		:=	OUT_OP.bGasTyp3_Act;
	xMsg1243.Reset		:=	TRUE;
	xMsg1243();
	bMsg1243			:=	xMsg1243.Q;

	(* B1244 selection gas type 4  *)
	xMsg1244.Enable		:=	TRUE;
	xMsg1244.Set		:=	OUT_OP.bGasTyp4_Act;
	xMsg1244.Reset		:=	TRUE;
	xMsg1244();
	bMsg1244			:=	xMsg1244.Q;

	(* B1245 selection ign.point 1 *)
	xMsg1245.Enable		:=	TRUE;
	xMsg1245.Set		:=	OUT_OP.bGasTyp1_Act AND (IN_OP.iIdx_Gtyp_Dem = 1);
	xMsg1245.Reset		:=	TRUE;
	xMsg1245();
	bMsg1245			:=	xMsg1245.Q;

	(* B1246 selection ign.point 2 *)
	xMsg1246.Enable		:=	TRUE;
	xMsg1246.Set		:=	OUT_OP.bGasTyp2_Act;
	xMsg1246.Reset		:=	TRUE;
	xMsg1246();
	bMsg1246			:=	xMsg1246.Q;

	(* B1247 selection ign.point 3 *)
	xMsg1247.Enable		:=	TRUE;
	xMsg1247.Set		:=	OUT_OP.bGasTyp3_Act;
	xMsg1247.Reset		:=	TRUE;
	xMsg1247();
	bMsg1247			:=	xMsg1247.Q;

	(* B1248 selection ign.point 4 *)
	xMsg1248.Enable		:=	TRUE;
	xMsg1248.Set		:=	OUT_OP.bGasTyp4_Act;
	xMsg1248.Reset		:=	TRUE;
	xMsg1248();
	bMsg1248			:=	xMsg1248.Q;

	(* B2122 *)
	xMsg2122.Enable		:=	TRUE;//NOT(Para.bP_SetCorr_FreqDroop AND IN_OP.iSource_F_N_OffsSet = 1) AND NOT(Para.bP_SetCorr_extNoffset AND IN_OP.iSource_F_N_OffsSet = 2);
	xMsg2122.Set		:=	xOpMode.NetP;
	xMsg2122.Reset		:=	TRUE;
	xMsg2122();
	bMsg2122			:=	xMsg2122.Q;

	(* B2123 *)
	xMsg2123.Enable		:=	TRUE;
	xMsg2123.Set		:=	xOpMode.Island;
	xMsg2123.Reset		:=	TRUE;
	xMsg2123();
	bMsg2123			:=	xMsg2123.Q;

	(* B2124 *)
	xMsg2124.Enable		:=	TRUE;
	xMsg2124.Set		:=	xOpMode.Idle;
	xMsg2124.Reset		:=	TRUE;
	xMsg2124();
	bMsg2124			:=	xMsg2124.Q;

	(* B2875 Power reduction by crank case pressure  *)
	xMsg2875.Enable		:=	TRUE;
	xMsg2875.Set		:=	xPRed[_CC].Q;
	xMsg2875.Reset		:=	TRUE;
	xMsg2875();
	MM2VIS.bMsg2875		:= 	xMsg2875.Q;

	(* B2168 generator air inlet temperature power reduction  *)
	xMsg2168.Enable		:=	TRUE;
	xMsg2168.Set		:=	xPRed[_GIAT].Q;
	xMsg2168.Reset		:=	TRUE;
	xMsg2168();
	MM2VIS.bMsg2168		:= 	xMsg2168.Q;

	(* B2925 Warm Up Operation *)
	xMsg2925.Enable		:=	TRUE;
	xMsg2925.Set		:=	bWarmUpOperation;
	xMsg2925.Reset		:=	TRUE;
	xMsg2925();
	MM2VIS.bMsg2925		:=	xMsg2925.Q;

	(* B2961 Power reduction by Cylinder Peak Pressure Integrator *)
	xMsg2961.Enable		:=	TRUE;
	xMsg2961.Set		:=	xPRed[_CPP].Q;
	xMsg2961.Reset		:=	TRUE;
	xMsg2961();
	MM2VIS.bMsg2961		:=	xMsg2961.Q;

	(* B2982 Power reduction calorific value *)
	xMsg2982.Enable		:=	TRUE;
	xMsg2982.Set		:=	xPRed[_CV].Q;
	xMsg2982.Reset		:=	TRUE;
	xMsg2982();
	MM2VIS.bMsg2982		:=	xMsg2982.Q;

	(* B2989 Power reduction by Generator Power Factor *)
	xTOF_Msg2989(IN:= xPRed[_GPF].Q, PT := T#60s);

	xMsg2989.Enable		:=	TRUE;
	xMsg2989.Set		:=	xTOF_Msg2989.Q;
	xMsg2989.Reset		:=	TRUE;
	xMsg2989();
	MM2VIS.bMsg2989		:=	xMsg2989.Q;

	(* B2972 Power Mode on *)
	xMsg2972.Enable		:=	TRUE;
	xMsg2972.Set		:=	bMsg2972;
	xMsg2972.Reset		:=	TRUE;
	xMsg2972();
	MM2VIS.bMsg2972		:=	xMsg2972.Q;

	(* B2973 Power Mode off *)
	xMsg2973.Enable		:=	TRUE;
	xMsg2973.Set		:=	bMsg2973;
	xMsg2973.Reset		:=	TRUE;
	xMsg2973();
	MM2VIS.bMsg2973		:=	xMsg2973.Q;

	(* B2935 Power reduction by CAN communication failure for half or more SAFI or too many SAFI reboots *)
	xMsg2935.Enable		:=	TRUE;
	xMsg2935.Set		:=	xPRed[_SAErr].Q;
	xMsg2935.Reset		:=	TRUE;
	xMsg2935();
	MM2VIS.bMsg2935		:=	xMsg2935.Q;

	MM2VIS.bMsg2162	:=	xPRed[_Trafo].Q;
	MM2VIS.bMsg2167	:=	xPRed[_GenCB].Q;

	MM2VIS.bMsg9024	:=	bIsland_Speed; 	(* B9024 - Isolated operation - Speed / Isochronous Mode *)
	MM2VIS.bMsg9025	:=	bIsland_Droop; 	(* B9025 - Isolated operation - Droop Mode *)
	MM2VIS.bMsg9026	:=	bIsland_LSL; 	(* B9026 - Isolated operation - Load sharing line *)

	(* B1283 B1284 B1285 B1286 B1287 Loadstep X reached with 1% hysterese - TOF 60s *)
	MM2VIS.bMsg1283	:=	TOF_LimitSon_Gh[0].Q AND Para.bP_GhStep_Ena;
	MM2VIS.bMsg1284	:=	TOF_LimitSon_Gh[1].Q AND Para.bP_GhStep_Ena;
	MM2VIS.bMsg1285	:=	TOF_LimitSon_Gh[2].Q AND Para.bP_GhStep_Ena;
	MM2VIS.bMsg1286	:=	TOF_LimitSon_Gh[3].Q AND Para.bP_GhStep_Ena;
	MM2VIS.bMsg1287	:=	TOF_LimitSon_Gh[4].Q AND Para.bP_GhStep_Ena;

	(* Request mode switch OFF, ON, REMOTE operating messages *)
	MM2VIS.bMsg2983 := OUT_OP.iIdx_RSS = 0;		(* Request mode switch OFF *)
	MM2VIS.bMsg2984 := OUT_OP.iIdx_RSS = 1;		(* Request mode switch ON *)
	MM2VIS.bMsg2985 := OUT_OP.iIdx_RSS = 2;		(* Request mode switch REMOTE *)

	(* B9051 Droop Mode for Power Controller *)
	xMsg9051.Enable		:=	TRUE;
	xMsg9051.Set		:=	bMsg9051;//xOpMode.NetP AND Para.bP_SetCorr_FreqDroop AND IN_OP.iSource_F_N_OffsSet = 1;
	xMsg9051.Reset		:=	TRUE;
	xMsg9051();
	MM2VIS.bMsg9051		:=	xMsg9051.Q;

	(* B9052 external speed reference offset Mode for Power Controller *)
	xMsg9052.Enable		:=	TRUE;
	xMsg9052.Set		:=	bMsg9052;//xOpMode.NetP AND Para.bP_SetCorr_extNoffset AND IN_OP.iSource_F_N_OffsSet = 2;
	xMsg9052.Reset		:=	TRUE;
	xMsg9052();
	MM2VIS.bMsg9052		:=	xMsg9052.Q;

	(* B9061 Activation Speed Setpoint Reduction due to overload of engine  *)
	xMsg9061.Enable		:=	TRUE;
	xMsg9061.Set		:=	Para.bN_SpdSetRed_Overload;
	xMsg9061.Reset		:=	TRUE;
	xMsg9061();
	MM2VIS.bMsg9061		:=	xMsg9061.Q;

	(* B9062 Deactivation Speed Setpoint Reduction due to overload of engine *)
	xMsg9062.Enable		:=	TRUE;
	xMsg9062.Set		:=	NOT Para.bN_SpdSetRed_Overload;
	xMsg9062.Reset		:=	TRUE;
	xMsg9062();
	MM2VIS.bMsg9062		:=	xMsg9062.Q;

	(* B9063 Power setpoint input external (myPlant) *)
	xMsg9063.Enable		:=	TRUE;
	xMsg9063.Set		:=	(OUT_OP.iIdx_Pset_Type = 18);
	xMsg9063.Reset		:=	TRUE;
	xMsg9063();
	MM2VIS.bMsg9063		:=	xMsg9063.Q;

	(* B9064 Request module on (myPlant) *)
	xMsg9064.Enable		:=	TRUE;
	xMsg9064.Set		:=	MM2VIS.bReq_Dem[7] AND OUT_OP.bEng_Dem;
	xMsg9064.Reset		:=	TRUE;
	xMsg9064();
	MM2VIS.bMsg9064		:=	xMsg9064.Q;

	(* B9072 Power reduction by H2 content *)
	xMsg9072.Enable		:=	TRUE;
	xMsg9072.Set		:=	xPRed[_H2].Q;
	xMsg9072.Reset		:=	TRUE;
	xMsg9072();
	MM2VIS.bMsg9072		:=	xMsg9072.Q;

	(* B9075 power reduction by charge temp. after HP TC *)
	xMsg9075.Enable		:=	TRUE;
	xMsg9075.Set		:=	xPRed[_T2HP].Q;
	xMsg9075.Reset		:=	TRUE;
	xMsg9075();
	MM2VIS.bMsg9075		:=	xMsg9075.Q;

	(* B9076 power reduction by charge temp. after LP TC *)
	xMsg9076.Enable		:=	TRUE;
	xMsg9076.Set		:=	xPRed[_T2LP].Q;
	xMsg9076.Reset		:=	TRUE;
	xMsg9076();
	MM2VIS.bMsg9076		:=	xMsg9076.Q;

	(*---------------------------------------------------------------------------*)
	(* general alarms for further module operations *)
	bGnlTrip1   := OUT_OP.tOP2AB.bGnlTrip1   OR IN_OP.tAB2OP.bGnlTrip1;
	bGnlTrip2   := OUT_OP.tOP2AB.bGnlTrip2   OR IN_OP.tAB2OP.bGnlTrip2;
	bGnlTrip3   := OUT_OP.tOP2AB.bGnlTrip3   OR IN_OP.tAB2OP.bGnlTrip3;
	bGnlWarning := OUT_OP.tOP2AB.bGnlWarning OR IN_OP.tAB2OP.bGnlWarning;

	bGnlTrip	:=	bGnlTrip1 OR bGnlTrip2 OR bGnlTrip3;

(*******************************************************************************)
END_PROGRAM
```

#### MsgOPInit.st - OpState Messages Init
```iecst
(*******************************************************************************
Msg_VE	 			 alarms generation MM_ventilation

This code is confidential and proprietary to the INNIO Company.
It may not be used in any form, or reproduced in any manner,
without written permission of the INNIO Company.
Copyright, INNIO Company, 2021

Customized modifications: -
------------------------

History:
-------
V0.00.0	29.07.2011	lettenb.	new
V0.11.0	22.12.2021	Andre		added B2935 Power reduction by CAN communication failure for half or more SAFI or too many SAFI reboots

Instructions for use:
--------------------
1) declare alarm with function block "Msg"

2) use template to create a new alarm, substitue 0000 by message number:

	xMsg0000.Num		:=	0000;					alarm number
	xMsg0000.AmmSysAdr	:=  iAdrAmmBase2MM;			do not change
	xMsg0000.AmmOutAdr	:=  iAdrMM2AmmBase;			do not change

3) 	set alarm number

Outstandings:
------------
(*******************************************************************************)
PROGRAM _INIT

	iAdrAmmBase2MM		:=  ADR(IN_OP.tAB2OP);
	iAdrMM2AmmBase		:=  ADR(OUT_OP.tOP2AB);

	(*---------------------------------------------------------------------------*)

	xMsg1108.Num		:=	1108;
	xMsg1108.AmmInAdr	:=  iAdrAmmBase2MM;
	xMsg1108.AmmOutAdr	:=  iAdrMM2AmmBase;

	xMsg3506.Num		:=	3506;
	xMsg3506.AmmInAdr	:=  iAdrAmmBase2MM;
	xMsg3506.AmmOutAdr	:=  iAdrMM2AmmBase;

	xMsg2082.Num		:=	2082;
	xMsg2082.AmmInAdr	:=  iAdrAmmBase2MM;
	xMsg2082.AmmOutAdr	:=  iAdrMM2AmmBase;

	xMsg1188.Num		:=	1188;
	xMsg1188.AmmInAdr	:=  iAdrAmmBase2MM;
	xMsg1188.AmmOutAdr	:=  iAdrMM2AmmBase;

	xMsg2097.Num		:=	2097;
	xMsg2097.AmmInAdr	:=  iAdrAmmBase2MM;
	xMsg2097.AmmOutAdr	:=  iAdrMM2AmmBase;

	xMsg1225.Num		:=	1225;
	xMsg1225.AmmInAdr	:=  iAdrAmmBase2MM;
	xMsg1225.AmmOutAdr	:=  iAdrMM2AmmBase;

	xMsg1226.Num		:=	1226;
	xMsg1226.AmmInAdr	:=  iAdrAmmBase2MM;
	xMsg1226.AmmOutAdr	:=  iAdrMM2AmmBase;

	xMsg1227.Num		:=	1227;
	xMsg1227.AmmInAdr	:=  iAdrAmmBase2MM;
	xMsg1227.AmmOutAdr	:=  iAdrMM2AmmBase;

	xMsg1228.Num		:=	1228;
	xMsg1228.AmmInAdr	:=  iAdrAmmBase2MM;
	xMsg1228.AmmOutAdr	:=  iAdrMM2AmmBase;

	xMsg1229.Num		:=	1229;
	xMsg1229.AmmInAdr	:=  iAdrAmmBase2MM;
	xMsg1229.AmmOutAdr	:=  iAdrMM2AmmBase;

	xMsg1230.Num		:=	1230;
	xMsg1230.AmmInAdr	:=  iAdrAmmBase2MM;
	xMsg1230.AmmOutAdr	:=  iAdrMM2AmmBase;

	xMsg1231.Num		:=	1231;
	xMsg1231.AmmInAdr	:=  iAdrAmmBase2MM;
	xMsg1231.AmmOutAdr	:=  iAdrMM2AmmBase;

	xMsg1232.Num		:=	1232;
	xMsg1232.AmmInAdr	:=  iAdrAmmBase2MM;
	xMsg1232.AmmOutAdr	:=  iAdrMM2AmmBase;

	xMsg1233.Num		:=	1233;
	xMsg1233.AmmInAdr	:=  iAdrAmmBase2MM;
	xMsg1233.AmmOutAdr	:=  iAdrMM2AmmBase;

	xMsg1234.Num		:=	1234;
	xMsg1234.AmmInAdr	:=  iAdrAmmBase2MM;
	xMsg1234.AmmOutAdr	:=  iAdrMM2AmmBase;

	xMsg1237.Num		:=	1237;
	xMsg1237.AmmInAdr	:=  iAdrAmmBase2MM;
	xMsg1237.AmmOutAdr	:=  iAdrMM2AmmBase;

	xMsg1238.Num		:=	1238;
	xMsg1238.AmmInAdr	:=  iAdrAmmBase2MM;
	xMsg1238.AmmOutAdr	:=  iAdrMM2AmmBase;

	xMsg1241.Num		:=	1241;
	xMsg1241.AmmInAdr	:=  iAdrAmmBase2MM;
	xMsg1241.AmmOutAdr	:=  iAdrMM2AmmBase;

	xMsg1242.Num		:=	1242;
	xMsg1242.AmmInAdr	:=  iAdrAmmBase2MM;
	xMsg1242.AmmOutAdr	:=  iAdrMM2AmmBase;

	xMsg1243.Num		:=	1243;
	xMsg1243.AmmInAdr	:=  iAdrAmmBase2MM;
	xMsg1243.AmmOutAdr	:=  iAdrMM2AmmBase;

	xMsg1244.Num		:=	1244;
	xMsg1244.AmmInAdr	:=  iAdrAmmBase2MM;
	xMsg1244.AmmOutAdr	:=  iAdrMM2AmmBase;

	xMsg1245.Num		:=	1245;
	xMsg1245.AmmInAdr	:=  iAdrAmmBase2MM;
	xMsg1245.AmmOutAdr	:=  iAdrMM2AmmBase;

	xMsg1246.Num		:=	1246;
	xMsg1246.AmmInAdr	:=  iAdrAmmBase2MM;
	xMsg1246.AmmOutAdr	:=  iAdrMM2AmmBase;

	xMsg1247.Num		:=	1247;
	xMsg1247.AmmInAdr	:=  iAdrAmmBase2MM;
	xMsg1247.AmmOutAdr	:=  iAdrMM2AmmBase;

	xMsg1248.Num		:=	1248;
	xMsg1248.AmmInAdr	:=  iAdrAmmBase2MM;
	xMsg1248.AmmOutAdr	:=  iAdrMM2AmmBase;

	xMsg2122.Num		:=	2122;
	xMsg2122.AmmInAdr	:=  iAdrAmmBase2MM;
	xMsg2122.AmmOutAdr	:=  iAdrMM2AmmBase;

	xMsg2123.Num		:=	2123;
	xMsg2123.AmmInAdr	:=  iAdrAmmBase2MM;
	xMsg2123.AmmOutAdr	:=  iAdrMM2AmmBase;

	xMsg2124.Num		:=	2124;
	xMsg2124.AmmInAdr	:=  iAdrAmmBase2MM;
	xMsg2124.AmmOutAdr	:=  iAdrMM2AmmBase;

	xMsg2125.Num		:=	2125;
	xMsg2125.AmmInAdr	:=  iAdrAmmBase2MM;
	xMsg2125.AmmOutAdr	:=  iAdrMM2AmmBase;

	xMsg2126.Num		:=	2126;
	xMsg2126.AmmInAdr	:=  iAdrAmmBase2MM;
	xMsg2126.AmmOutAdr	:=  iAdrMM2AmmBase;

	xMsg2127.Num		:=	2127;
	xMsg2127.AmmInAdr	:=  iAdrAmmBase2MM;
	xMsg2127.AmmOutAdr	:=  iAdrMM2AmmBase;

	xMsg2128.Num		:=	2128;
	xMsg2128.AmmInAdr	:=  iAdrAmmBase2MM;
	xMsg2128.AmmOutAdr	:=  iAdrMM2AmmBase;

	xMsg2129.Num		:=	2129;
	xMsg2129.AmmInAdr	:=  iAdrAmmBase2MM;
	xMsg2129.AmmOutAdr	:=  iAdrMM2AmmBase;

	xMsg2130.Num		:=	2130;
	xMsg2130.AmmInAdr	:=  iAdrAmmBase2MM;
	xMsg2130.AmmOutAdr	:=  iAdrMM2AmmBase;

	xMsg2131.Num		:=	2131;
	xMsg2131.AmmInAdr	:=  iAdrAmmBase2MM;
	xMsg2131.AmmOutAdr	:=  iAdrMM2AmmBase;

	xMsg2132.Num		:=	2132;
	xMsg2132.AmmInAdr	:=  iAdrAmmBase2MM;
	xMsg2132.AmmOutAdr	:=  iAdrMM2AmmBase;

	xMsg2140.Num		:=	2140;
	xMsg2140.AmmInAdr	:=  iAdrAmmBase2MM;
	xMsg2140.AmmOutAdr	:=  iAdrMM2AmmBase;

	xMsg2143.Num		:=	2143;
	xMsg2143.AmmInAdr	:=  iAdrAmmBase2MM;
	xMsg2143.AmmOutAdr	:=  iAdrMM2AmmBase;

	xMsg2144.Num		:=	2144;
	xMsg2144.AmmInAdr	:=  iAdrAmmBase2MM;
	xMsg2144.AmmOutAdr	:=  iAdrMM2AmmBase;

	xMsg2146.Num		:=	2146;
	xMsg2146.AmmInAdr	:=  iAdrAmmBase2MM;
	xMsg2146.AmmOutAdr	:=  iAdrMM2AmmBase;

	xMsg2147.Num		:=	2147;
	xMsg2147.AmmInAdr	:=  iAdrAmmBase2MM;
	xMsg2147.AmmOutAdr	:=  iAdrMM2AmmBase;

	xMsg2148.Num		:=	2148;
	xMsg2148.AmmInAdr	:=  iAdrAmmBase2MM;
	xMsg2148.AmmOutAdr	:=  iAdrMM2AmmBase;

	xMsg2149.Num		:=	2149;
	xMsg2149.AmmInAdr	:=  iAdrAmmBase2MM;
	xMsg2149.AmmOutAdr	:=  iAdrMM2AmmBase;

	xMsg2150.Num		:=	2150;
	xMsg2150.AmmInAdr	:=  iAdrAmmBase2MM;
	xMsg2150.AmmOutAdr	:=  iAdrMM2AmmBase;

	xMsg2152.Num		:=	2152;
	xMsg2152.AmmInAdr	:=  iAdrAmmBase2MM;
	xMsg2152.AmmOutAdr	:=  iAdrMM2AmmBase;

	xMsg2153.Num		:=	2153;
	xMsg2153.AmmInAdr	:=  iAdrAmmBase2MM;
	xMsg2153.AmmOutAdr	:=  iAdrMM2AmmBase;

	xMsg2154.Num		:=	2154;
	xMsg2154.AmmInAdr	:=  iAdrAmmBase2MM;
	xMsg2154.AmmOutAdr	:=  iAdrMM2AmmBase;

	xMsg2155.Num		:=	2155;
	xMsg2155.AmmInAdr	:=  iAdrAmmBase2MM;
	xMsg2155.AmmOutAdr	:=  iAdrMM2AmmBase;

	xMsg2158.Num		:=	2158;
	xMsg2158.AmmInAdr	:=  iAdrAmmBase2MM;
	xMsg2158.AmmOutAdr	:=  iAdrMM2AmmBase;

	xMsg2159.Num		:=	2159;
	xMsg2159.AmmInAdr	:=  iAdrAmmBase2MM;
	xMsg2159.AmmOutAdr	:=  iAdrMM2AmmBase;

	xMsg2160.Num		:=	2160;
	xMsg2160.AmmInAdr	:=  iAdrAmmBase2MM;
	xMsg2160.AmmOutAdr	:=  iAdrMM2AmmBase;

	xMsg2161.Num		:=	2161;
	xMsg2161.AmmInAdr	:=  iAdrAmmBase2MM;
	xMsg2161.AmmOutAdr	:=  iAdrMM2AmmBase;

	xMsg2163.Num		:=	2163;
	xMsg2163.AmmInAdr	:=  iAdrAmmBase2MM;
	xMsg2163.AmmOutAdr	:=  iAdrMM2AmmBase;

	xMsg2164.Num		:=	2164;
	xMsg2164.AmmInAdr	:=  iAdrAmmBase2MM;
	xMsg2164.AmmOutAdr	:=  iAdrMM2AmmBase;

	xMsg2168.Num 		:= 	2168;
	xMsg2168.AmmInAdr 	:= iAdrAmmBase2MM;
	xMsg2168.AmmOutAdr 	:= iAdrMM2AmmBase;

	xMsg2169.Num		:=	2169;
	xMsg2169.AmmInAdr	:=  iAdrAmmBase2MM;
	xMsg2169.AmmOutAdr	:=  iAdrMM2AmmBase;

	xMsg2170.Num		:=	2170;
	xMsg2170.AmmInAdr	:=  iAdrAmmBase2MM;
	xMsg2170.AmmOutAdr	:=  iAdrMM2AmmBase;

	xMsg2803.Num		:=	2803;
	xMsg2803.AmmInAdr	:=  iAdrAmmBase2MM;
	xMsg2803.AmmOutAdr	:=  iAdrMM2AmmBase;

	xMsg2875.Num 		:= 	2875;
	xMsg2875.AmmInAdr 	:= iAdrAmmBase2MM;
	xMsg2875.AmmOutAdr 	:= iAdrMM2AmmBase;

	xMsg2925.Num		:=	2925;
	xMsg2925.AmmInAdr	:=  iAdrAmmBase2MM;
	xMsg2925.AmmOutAdr	:=  iAdrMM2AmmBase;

	xMsg2936.Num		:=	2936;
	xMsg2936.AmmInAdr	:=  iAdrAmmBase2MM;
	xMsg2936.AmmOutAdr	:=  iAdrMM2AmmBase;

	xMsg2961.Num 		:= 	2961;
	xMsg2961.AmmInAdr 	:=  iAdrAmmBase2MM;
	xMsg2961.AmmOutAdr 	:=  iAdrMM2AmmBase;

	xMsg3229.Num		:=	3229;
	xMsg3229.AmmInAdr	:=  iAdrAmmBase2MM;
	xMsg3229.AmmOutAdr	:=  iAdrMM2AmmBase;

	xMsg3230.Num		:=	3230;
	xMsg3230.AmmInAdr	:=  iAdrAmmBase2MM;
	xMsg3230.AmmOutAdr	:=  iAdrMM2AmmBase;

	xMsg3231.Num		:=	3231;
	xMsg3231.AmmInAdr	:=  iAdrAmmBase2MM;
	xMsg3231.AmmOutAdr	:=  iAdrMM2AmmBase;

	xMsg2982.Num		:=	2982;
	xMsg2982.AmmInAdr	:=  iAdrAmmBase2MM;
	xMsg2982.AmmOutAdr	:=  iAdrMM2AmmBase;

	xMsg2989.Num		:=	2989;
	xMsg2989.AmmInAdr	:=  iAdrAmmBase2MM;
	xMsg2989.AmmOutAdr	:=  iAdrMM2AmmBase;

	xMsg9284.Num		:=	9284;
	xMsg9284.AmmInAdr	:=  iAdrAmmBase2MM;
	xMsg9284.AmmOutAdr	:=  iAdrMM2AmmBase;

	xMsg2972.Num		:=	2972;
	xMsg2972.AmmInAdr	:=  iAdrAmmBase2MM;
	xMsg2972.AmmOutAdr	:=  iAdrMM2AmmBase;

	xMsg2973.Num		:=	2973;
	xMsg2973.AmmInAdr	:=  iAdrAmmBase2MM;
	xMsg2973.AmmOutAdr	:=  iAdrMM2AmmBase;

	xMsg9051.Num		:=	9051;
	xMsg9051.AmmInAdr	:=  iAdrAmmBase2MM;
	xMsg9051.AmmOutAdr	:=  iAdrMM2AmmBase;

	xMsg9052.Num		:=	9052;
	xMsg9052.AmmInAdr	:=  iAdrAmmBase2MM;
	xMsg9052.AmmOutAdr	:=  iAdrMM2AmmBase;

	xMsg9061.Num		:=	9061;
	xMsg9061.AmmInAdr	:=  iAdrAmmBase2MM;
	xMsg9061.AmmOutAdr	:=  iAdrMM2AmmBase;

	xMsg9062.Num		:=	9062;
	xMsg9062.AmmInAdr	:=  iAdrAmmBase2MM;
	xMsg9062.AmmOutAdr	:=  iAdrMM2AmmBase;

	xMsg9063.Num		:=	9063;
	xMsg9063.AmmInAdr	:=  iAdrAmmBase2MM;
	xMsg9063.AmmOutAdr	:=  iAdrMM2AmmBase;

	xMsg9064.Num		:=	9064;
	xMsg9064.AmmInAdr	:=  iAdrAmmBase2MM;
	xMsg9064.AmmOutAdr	:=  iAdrMM2AmmBase;

	xMsg2935.Num		:=	2935;
	xMsg2935.AmmInAdr	:=  iAdrAmmBase2MM;
	xMsg2935.AmmOutAdr	:=  iAdrMM2AmmBase;

	xMsg9072.Num		:=	9072;
	xMsg9072.AmmInAdr	:=  iAdrAmmBase2MM;
	xMsg9072.AmmOutAdr	:=  iAdrMM2AmmBase;

	xMsg9075.Num		:=	9075;
	xMsg9075.AmmInAdr	:=  iAdrAmmBase2MM;
	xMsg9075.AmmOutAdr	:=  iAdrMM2AmmBase;

	xMsg9076.Num		:=	9076;
	xMsg9076.AmmInAdr	:=  iAdrAmmBase2MM;
	xMsg9076.AmmOutAdr	:=  iAdrMM2AmmBase;

END_PROGRAM
```

#### MsgOP.var
```iecst
VAR
	iAdrMM2AmmBase : UDINT;
	iAdrAmmBase2MM : UDINT;
	xTOF_Msg2130 : TOF;
	xTOF_Msg2152 : TOF;
	xTOF_Msg2153 : TOF;
	xTOF_Msg2154 : TOF;
	xTOF_Msg2989 : TOF;
	xMsg1225 : Msg;
	xMsg1226 : Msg;
	xMsg1227 : Msg;
	xMsg1228 : Msg;
	xMsg1229 : Msg;
	xMsg1230 : Msg;
	xMsg1231 : Msg;
	xMsg1232 : Msg;
	xMsg1233 : Msg;
	xMsg1234 : Msg;
	xMsg1237 : Msg;
	xMsg1238 : Msg;
	xMsg1241 : Msg;
	xMsg1242 : Msg;
	xMsg1243 : Msg;
	xMsg1244 : Msg;
	xMsg1245 : Msg;
	xMsg1246 : Msg;
	xMsg1247 : Msg;
	xMsg1248 : Msg;
	xMsg2122 : Msg;
	xMsg2123 : Msg;
	xMsg2124 : Msg;
	xMsg2125 : Msg;
	xMsg2126 : Msg;
	xMsg2127 : Msg;
	xMsg2128 : Msg;
	xMsg2129 : Msg;
	xMsg2130 : Msg;
	xMsg2131 : Msg;
	xMsg2132 : Msg;
	xMsg2140 : Msg;
	xMsg2143 : Msg;
	xMsg2144 : Msg;
	xMsg2146 : Msg;
	xMsg2147 : Msg;
	xMsg2148 : Msg;
	xMsg2149 : Msg;
	xMsg2150 : Msg;
	xMsg2152 : Msg;
	xMsg2153 : Msg;
	xMsg2154 : Msg;
	xMsg2155 : Msg;
	xMsg2158 : Msg;
	xMsg2159 : Msg;
	xMsg2160 : Msg;
	xMsg2161 : Msg;
	xMsg2163 : Msg;
	xMsg2164 : Msg;
	xMsg2170 : Msg;
	xMsg2169 : Msg;
	xMsg2803 : Msg;
	xMsg2936 : Msg;
	xMsg2961 : Msg;
	xMsg3229 : Msg;
	xMsg3230 : Msg;
	xMsg2982 : Msg;
	xMsg3231 : Msg;
	xMsg2875 : Msg;
	xMsg2168 : Msg;
	xMsg2925 : Msg;
	xMsg2989 : Msg;
	xMsg9284 : Msg;
	xMsg2972 : Msg;
	xMsg2973 : Msg;
	xMsg9051 : Msg;
	xMsg9052 : Msg;
	xMsg9061 : Msg;
	xMsg9062 : Msg;
	xMsg9063 : Msg;
	xMsg9064 : Msg;
	xMsg2935 : Msg;
	xMsg9072 : Msg;
	xMsg9075 : Msg;
	xMsg9076 : Msg;
END_VAR
```

### Program Logical/Opstate/VisOP (IEC) - Visualisation Communication
